// TIA Portal project "杨村程序" (V15.1)

(* hardware
DEVICE "S71500/ET200MP station_1"  S7-1500 station
   slot 0: "导轨_0"  Rack  6ES7 590-1***0-0AA0
   slot 1: "PLC_1"  CPU 1511-1 PN  6ES7 511-1AK02-0AB0  V2.6
      slot 3: "CPU 显示_1"  6ES7591-1AA00-0AA0
DEVICE "ET 200SP station_1"  ET 200SP-Station
   slot 0: "机架_0"  Rack  6ES5 710-8MAx1
   slot 0: "IO device_1"  IM 155-6 PN ST  6ES7 155-6AU01-0BN0  V4.1
   slot 1: "DI 16x24VDC ST_1"  DI 16x24VDC ST  6ES7 131-6BH01-0BA0  V0.0
      slot 1: "DI 16x24VDC ST_1"  DI 16x24VDC ST
   slot 2: "DI 16x24VDC ST_2"  DI 16x24VDC ST  6ES7 131-6BH01-0BA0  V0.0
      slot 1: "DI 16x24VDC ST_2"  DI 16x24VDC ST
   slot 3: "DI 16x24VDC ST_3"  DI 16x24VDC ST  6ES7 131-6BH01-0BA0  V0.0
      slot 1: "DI 16x24VDC ST_3"  DI 16x24VDC ST
   slot 4: "DI 16x24VDC ST_4"  DI 16x24VDC ST  6ES7 131-6BH01-0BA0  V0.0
      slot 1: "DI 16x24VDC ST_4"  DI 16x24VDC ST
   slot 5: "DQ 16x24VDC/0.5A ST_1"  DQ 16x24VDC/0.5A ST  6ES7 132-6BH01-0BA0  V0.0
      slot 1: "DQ 16x24VDC/0.5A ST_1"  DQ 16x24VDC/0.5A ST
   slot 6: "DQ 16x24VDC/0.5A ST_2"  DQ 16x24VDC/0.5A ST  6ES7 132-6BH01-0BA0  V0.0
      slot 1: "DQ 16x24VDC/0.5A ST_2"  DQ 16x24VDC/0.5A ST
   slot 7: "AI 8xI 2-,4-wire BA_1"  AI 8xI 2-,4-wire BA  6ES7 134-6GF00-0AA1  V1.0
      slot 1: "AI 8xI 2-,4-wire BA_1"  AI 8xI 2-,4-wire BA
   slot 8: "AI 8xI 2-,4-wire BA_2"  AI 8xI 2-,4-wire BA  6ES7 134-6GF00-0AA1  V1.0
      slot 1: "AI 8xI 2-,4-wire BA_2"  AI 8xI 2-,4-wire BA
   slot 9: "AI 8xI 2-,4-wire BA_3"  AI 8xI 2-,4-wire BA  6ES7 134-6GF00-0AA1  V1.0
      slot 1: "AI 8xI 2-,4-wire BA_3"  AI 8xI 2-,4-wire BA
   slot 10: "AI 8xI 2-,4-wire BA_4"  AI 8xI 2-,4-wire BA  6ES7 134-6GF00-0AA1  V1.0
      slot 1: "AI 8xI 2-,4-wire BA_4"  AI 8xI 2-,4-wire BA
   slot 11: "AQ 4xU/I ST_1"  AQ 4xU/I ST  6ES7 135-6HD00-0BA1  V1.1
      slot 1: "AQ 4xU/I ST_1"  AQ 4xU/I ST
   slot 12: "CM PtP_1"  CM PtP  6ES7 137-6AA00-0BA0  V1.0
      slot 1: "CM PtP_1"  CM PtP Sub
   slot 13: "服务器模块_1"  Server module  6ES7 193-6PA00-0AA0  V1.1
      slot 1: "服务器模块_1"  Server module
   slot 127: "BA 2xRJ45"  BA 2xRJ45  6ES7 193-6AR00-0AA0  V0.0
      slot 1: "Port_1"  X1 P1 R  6ES7 193-6AR00-0AA0  V0.0
      slot 2: "Port_2"  X1 P2 R  6ES7 193-6AR00-0AA0  V0.0
*)

// ===== PLC "PLC_1"  CPU 1511-1 PN =====

VAR_GLOBAL   // PLC tag table "默认变量表"
   "P1_HS" AT %IW8 : Int;
   "P2_HS" AT %IW10 : Int;
   "P3_GS" AT %IW12 : Int;
   "P4_GSFJK" AT %IW14 : Int;
   "P5_HSFJK" AT %IW16 : Int;
   "P6_GSCN" AT %IW18 : Int;
   "P7_HSCN" AT %IW20 : Int;
   "P1_能源站进站泵前压力" AT %MD100 : Real;
   "P2_能源站进站泵后压力" AT %MD104 : Real;
   "P3_能源站出站压力" AT %MD108 : Real;
   "P4_副井口供水压力" AT %MD112 : Real;
   "P5_副井口回水压力" AT %MD116 : Real;
   "P6_采暖供水压力" AT %MD120 : Real;
   "P7_采暖回水压力" AT %MD124 : Real;
   "T1_HS" AT %IW24 : Int;
   "T2_GS" AT %IW26 : Int;
   "T3_HSFJK1" AT %IW28 : Int;
   "T4_GSFJK1" AT %IW30 : Int;
   "T5_HSFJK2" AT %IW32 : Int;
   "T6_GSFJK2" AT %IW34 : Int;
   "T7_GSFJK" AT %IW36 : Int;
   "T8_HSFJK" AT %IW38 : Int;
   "T9_GSCN" AT %IW40 : Int;
   "T10_HSCN" AT %IW42 : Int;
   "T11_FJK_HJ" AT %IW44 : Int;
   "T12_SW_HJ" AT %IW46 : Int;
   "T1_能源站进站温度" AT %MD128 : Real;
   "T2_能源站出站温度" AT %MD132 : Real;
   "T3_副井口换热器一次进水" AT %MD136 : Real;
   "T4_副井口换热器一次出水" AT %MD140 : Real;
   "T5_副井口换热器二次进水" AT %MD144 : Real;
   "T6_副井口换热器二次出水" AT %MD148 : Real;
   "T7_副井口供水" AT %MD152 : Real;
   "T8_副井口回水" AT %MD156 : Real;
   "T9_采暖供水" AT %MD160 : Real;
   "T10_采暖回水" AT %MD164 : Real;
   "T11_副井口环境温度" AT %MD168 : Real;
   "T12_环境温度" AT %MD172 : Real;
   "隔离水泵运行频率" AT %MD176 : Real;
   "隔离水泵设定频率" AT %MD180 : Real;
   "MF1_ReadValue" AT %IW70 : Int;
   "System_Byte" AT %MB1 : Byte;
   "FirstScan" AT %M1.0 : Bool;
   "DiagStatusUpdate" AT %M1.1 : Bool;
   "AlwaysTRUE" AT %M1.2 : Bool;
   "AlwaysFALSE" AT %M1.3 : Bool;
   "Clock_Byte" AT %MB0 : Byte;
   "Clock_10Hz" AT %M0.0 : Bool;
   "Clock_5Hz" AT %M0.1 : Bool;
   "Clock_2.5Hz" AT %M0.2 : Bool;
   "Clock_2Hz" AT %M0.3 : Bool;
   "Clock_1.25Hz" AT %M0.4 : Bool;
   "Clock_1Hz" AT %M0.5 : Bool;
   "Clock_0.625Hz" AT %M0.6 : Bool;
   "Clock_0.5Hz" AT %M0.7 : Bool;
   "RM1_瞬时流量" AT %MD200 : Real;
   "RM1_瞬时热流量" AT %MD204 : Real;
   "RM1_累计热量" AT %MD208 : Real;
   "RM1_入口温度" AT %MD212 : Real;
   "RM1_出口温度" AT %MD216 : Real;
   "RM2_瞬时流量" AT %MD220 : Real;
   "RM2_瞬时热流量" AT %MD224 : Real;
   "RM2_累计热量" AT %MD228 : Real;
   "RM2_入口温度" AT %MD232 : Real;
   "RM2_出口温度" AT %MD236 : Real;
   "RM3_瞬时流量" AT %MD240 : Real;
   "RM3_瞬时热流量" AT %MD244 : Real;
   "RM3_累计热量" AT %MD248 : Real;
   "RM3_入口温度" AT %MD252 : Real;
   "RM3_出口温度" AT %MD256 : Real;
   "RM4_瞬时流量" AT %MD260 : Real;
   "RM4_瞬时热流量" AT %MD264 : Real;
   "RM4_累计热量" AT %MD268 : Real;
   "RM4_入口温度" AT %MD272 : Real;
   "RM4_出口温度" AT %MD276 : Real;
   "RM5_瞬时流量" AT %MD280 : Real;
   "RM5_瞬时热流量" AT %MD284 : Real;
   "RM5_累计热量" AT %MD288 : Real;
   "RM5_入口温度" AT %MD292 : Real;
   "RM5_出口温度" AT %MD296 : Real;
   "#1隔离泵手自状态反馈" AT %I0.0 : Bool;
   "#1隔离泵变频运行反馈" AT %I0.1 : Bool;
   "#1隔离泵变频故障反馈" AT %I0.2 : Bool;
   "#2隔离泵手自状态反馈" AT %I0.4 : Bool;
   "#2隔离泵软起运行反馈" AT %I0.5 : Bool;
   "#2隔离泵软起故障反馈" AT %I0.6 : Bool;
   "旁通电动阀手自状态反馈" AT %I1.0 : Bool;
   "#1电动阀全开反馈" AT %I1.1 : Bool;
   "#1电动阀全关反馈" AT %I1.2 : Bool;
   "#2电动阀全开反馈" AT %I1.3 : Bool;
   "#2电动阀全关反馈" AT %I1.4 : Bool;
   "#1进站水流开关状态" AT %I1.5 : Bool;
   "#2副井口水流开关状态" AT %I1.6 : Bool;
   "#3采暖水流开关状态" AT %I1.7 : Bool;
   "采暖循环泵手自状态反馈" AT %I2.0 : Bool;
   "#1采暖循环泵运行反馈" AT %I2.1 : Bool;
   "#2采暖循环泵运行反馈" AT %I2.2 : Bool;
   "#1采暖循环泵故障反馈" AT %I2.3 : Bool;
   "#2采暖循环泵故障反馈" AT %I2.4 : Bool;
   "副井口循环泵手自状态反馈" AT %I3.0 : Bool;
   "#1副井口循环泵运行反馈" AT %I3.1 : Bool;
   "#2副井口循环泵运行反馈" AT %I3.2 : Bool;
   "#3副井口循环泵运行反馈" AT %I3.3 : Bool;
   "供热补水泵手自状态反馈" AT %I4.0 : Bool;
   "#1供热补水泵运行反馈" AT %I4.1 : Bool;
   "#2供热补水泵运行反馈" AT %I4.2 : Bool;
   "矿区补水泵手自状态反馈" AT %I4.3 : Bool;
   "#1矿区补水泵运行反馈" AT %I4.4 : Bool;
   "#2矿区补水泵运行反馈" AT %I4.5 : Bool;
   "增压泵手自状态反馈" AT %I2.5 : Bool;
   "增加泵软起运行反馈" AT %I2.6 : Bool;
   "增压泵软起故障反馈" AT %I2.7 : Bool;
   "#1隔离水泵启停控制" AT %Q0.0 : Bool;
   "#2隔离水泵启停控制" AT %Q0.1 : Bool;
   "#1热泵机组旁通阀开控制" AT %Q0.2 : Bool;
   "#1热泵机组旁通阀关控制" AT %Q0.3 : Bool;
   "#2热泵机组旁通阀开控制" AT %Q0.4 : Bool;
   "#2热泵机组旁通阀关控制" AT %Q0.5 : Bool;
   "#1采暖泵启停控制" AT %Q0.6 : Bool;
   "#2采暖泵启停控制" AT %Q0.7 : Bool;
   "副井口#1采暖循环泵控制" AT %Q1.0 : Bool;
   "副井口#2采暖循环泵控制" AT %Q1.1 : Bool;
   "副井口#3采暖循环泵控制" AT %Q1.2 : Bool;
   "供热#1补水泵控制" AT %Q1.3 : Bool;
   "供热#2补水泵控制" AT %Q1.4 : Bool;
   "矿区#1补水泵控制" AT %Q1.5 : Bool;
   "矿区#2补水泵控制" AT %Q1.6 : Bool;
   "蜂鸣报警输出" AT %Q1.7 : Bool;
   "增压泵启停控制" AT %Q2.4 : Bool;
   "M_采暖#1泵手动启停" AT %M10.0 : Bool;
   "M_采暖#2泵手动启停" AT %M10.1 : Bool;
   "M_增压泵手动启停" AT %M10.2 : Bool;
   "M_副井口#1泵手动启停" AT %M10.3 : Bool;
   "M_副井口#2泵手动启停" AT %M10.4 : Bool;
   "M_副井口#3泵手动启停" AT %M10.5 : Bool;
   "M_隔离#1泵手动启停" AT %M10.6 : Bool;
   "M_隔离#2泵手动启停" AT %M10.7 : Bool;
   "M_供热补水#1泵手动启停" AT %M11.0 : Bool;
   "M_供热补水#2泵手动启停" AT %M11.1 : Bool;
   "M_矿区补水#1泵手动启停" AT %M11.2 : Bool;
   "M_矿区补水#2泵手动启停" AT %M11.3 : Bool;
   "M_旁通#1阀手动开关" AT %M11.4 : Bool;
   "M_旁通#2阀手动开关" AT %M11.5 : Bool;
   "M_电磁阀#1手动开关" AT %M11.6 : Bool;
   "S_循环水泵投入退出" AT %M2.0 : Bool;
   "水箱电磁阀启停控制" AT %Q3.4 : Bool;
   "Tag_2" AT %M20.1 : Bool;
   "Tag_3" AT %M20.0 : Bool;
   "Tag_4" AT %M20.2 : Bool;
   "Tag_5" AT %M20.3 : Bool;
   "Tag_6" AT %M20.4 : Bool;
   "Tag_7" AT %M20.5 : Bool;
   "Tag_8" AT %M20.6 : Bool;
   "Tag_9" AT %M20.7 : Bool;
   "Tag_10" AT %M21.0 : Bool;
   "Tag_11" AT %M21.1 : Bool;
   "Tag_12" AT %M21.2 : Bool;
   "Tag_13" AT %M21.3 : Bool;
   "Tag_14" AT %M21.4 : Bool;
   "Tag_15" AT %M21.5 : Bool;
   "Tag_16" AT %M21.6 : Bool;
   "Tag_17" AT %M21.7 : Bool;
   "Tag_18" AT %M22.0 : Bool;
   "Tag_19" AT %M22.1 : Bool;
   "Tag_20" AT %M22.2 : Bool;
   "Tag_21" AT %M22.3 : Bool;
   "Tag_22" AT %M22.4 : Bool;
   "Tag_23" AT %M22.5 : Bool;
   "Tag_24" AT %M22.6 : Bool;
   "Tag_25" AT %M22.7 : Bool;
   "Tag_26" AT %M23.0 : Bool;
   "Tag_27" AT %M23.1 : Bool;
   "Tag_28" AT %M23.2 : Bool;
   "Tag_29" AT %M23.3 : Bool;
   "Tag_30" AT %M23.4 : Bool;
   "Tag_31" AT %M23.5 : Bool;
   "系统运行天数" AT %MW90 : UInt;
   "系统运行小时" AT %MW92 : UInt;
   "系统运行分钟" AT %MW94 : UInt;
   "M_副井口排污阀手动开关" AT %M11.7 : Bool;
   "Tag_33" AT %M23.6 : Bool;
   "Tag_34" AT %M23.7 : Bool;
   "温度传感器上限" AT %MD310 : Real;
   "温度传感器下限" AT %MD314 : Real;
   "压力传感器上限" AT %MD318 : Real;
   "压力传感器下限" AT %MD322 : Real;
   "#1吸收式热泵启停指令" AT %MW326 : UInt;
   "#2吸收式热泵启停指令" AT %MW328 : UInt;
   "M_热泵 #1手动开关" AT %M12.0 : Bool;
   "M_热泵 #2手动开关" AT %M12.1 : Bool;
   "Tag_1" AT %M24.0 : Bool;
   "Tag_35" AT %M24.1 : Bool;
   "Tag_36" AT %M24.2 : Bool;
   "Tag_37" AT %M24.3 : Bool;
   "变频器频率上限" AT %MD330 : Real;
   "变频器频率下限" AT %MD334 : Real;
   "MF1_WriteFValue" AT %QW4 : Int;
   "#1热泵热网水进口温度" AT %MD340 : Real;
   "#1热泵热网水出口温度" AT %MD344 : Real;
   "#1热泵热源水进口温度" AT %MD348 : Real;
   "#1热泵热源水出口温度" AT %MD352 : Real;
   "#1热泵驱动热水进口温度" AT %MD356 : Real;
   "#1热泵驱动热水出口温度" AT %MD360 : Real;
   "#2热泵热网水进口温度" AT %MD364 : Real;
   "#2热泵热网水出口温度" AT %MD368 : Real;
   "#2热泵热源水进口温度" AT %MD372 : Real;
   "#2热泵热源水出口温度" AT %MD376 : Real;
   "#2热泵驱动热水进口温度" AT %MD380 : Real;
   "#2热泵驱动热水出口温度" AT %MD384 : Real;
   "国焦侧供水温度" AT %MD388 : Real;
   "国焦侧回水温度" AT %MD392 : Real;
   "国焦侧氨水进水温度" AT %MD396 : Real;
   "国焦侧氨水回水温度" AT %MD400 : Real;
   "国焦侧蒸汽瞬时流量" AT %MD404 : Real;
   "供热补水压力上限" AT %MD408 : Real;
   "供热补水压力下限" AT %MD412 : Real;
   "矿区补水压力上限" AT %MD416 : Real;
   "矿区补水压力下限" AT %MD420 : Real;
   "M_补水泵手自投入退出" AT %M2.1 : Bool;
   "Tag_38" AT %M24.5 : Bool;
   "Tag_39" AT %M24.6 : Bool;
   "Tag_40" AT %M24.7 : Bool;
   "Tag_41" AT %M25.0 : Bool;
   "Tag_42" AT %M25.1 : Bool;
   "Tag_43" AT %M25.2 : Bool;
   "Tag_44" AT %M25.3 : Bool;
   "Tag_45" AT %M25.4 : Bool;
   "补水参数设置错误" AT %M50.6 : Bool;
   "水箱液位" AT %MD424 : Real;
   "H_Yewei" AT %IW56 : Int;
   "电加热管道AP7电源合闸反馈" AT %I3.4 : Bool;
   "电加热管道AP7电源分闸反馈" AT %I3.5 : Bool;
   "电加热管道AP7电源故障反馈" AT %I3.6 : Bool;
   "电加热管道AP8电源合闸反馈" AT %I5.4 : Bool;
   "电加热管道AP8电源分闸反馈" AT %I5.5 : Bool;
   "电加热管道AP8电源故障反馈" AT %I5.6 : Bool;
   "#2采暖排污阀关控制" AT %Q3.3 : Bool;
   "#2采暖排污阀开控制" AT %Q3.2 : Bool;
   "#1副井口排污阀关控制" AT %Q3.1 : Bool;
   "#1副井口排污阀开控制" AT %Q3.0 : Bool;
   "#1副井口排污阀开反馈" AT %I5.0 : Bool;
   "M_采暖排污阀手动开关" AT %M12.2 : Bool;
   "Tag_47" AT %M25.5 : Bool;
   "Tag_48" AT %M25.6 : Bool;
   "Tag_49" AT %M25.7 : Bool;
   "Tag_50" AT %M26.0 : Bool;
   "报警_水箱液位低" AT %M50.0 : Bool;
   "报警_水箱液位高" AT %M50.1 : Bool;
   "供热补水泵#1投入" AT %M3.1 : Bool;
   "modbus_Step" AT %MW56 : UInt;
   "供热补水泵#2投入" AT %M3.2 : Bool;
   "矿区补水泵#1投入" AT %M3.3 : Bool;
   "矿区补水泵#2投入" AT %M3.4 : Bool;
   "#1副井口排污阀关反馈" AT %I5.1 : Bool;
   "#2采暖排污阀开反馈" AT %I5.2 : Bool;
   "#2采暖排污阀关反馈" AT %I5.3 : Bool;
   "#1热泵启动控制" AT %Q2.0 : Bool;
   "#1热泵急停控制" AT %Q2.1 : Bool;
   "#2热泵启动控制" AT %Q2.2 : Bool;
   "#2热泵急停控制" AT %Q2.3 : Bool;
   "P1_能源站进站泵前压力_工程值" AT %MD428 : Real;
   "P2_能源站进站泵后压力_工程值" AT %MD432 : Real;
   "P3_能源站出站压力_工程值" AT %MD436 : Real;
   "P4_副井口供水压力_工程值" AT %MD440 : Real;
   "P5_副井口回水压力_工程值" AT %MD444 : Real;
   "P6_采暖供水压力_工程值" AT %MD448 : Real;
   "P7_采暖回水压力_工程值" AT %MD452 : Real;
   "T1_能源站进站温度_工程值" AT %MD456 : Real;
   "T2_能源站出站温度_工程值" AT %MD460 : Real;
   "T3_副井口换热器一次进水_工程值" AT %MD464 : Real;
   "T4_副井口换热器一次出水_工程值" AT %MD468 : Real;
   "T5_副井口换热器二次进水_工程值" AT %MD472 : Real;
   "T6_副井口换热器二次出水_工程值" AT %MD476 : Real;
   "T7_副井口供水_工程值" AT %MD480 : Real;
   "T8_副井口回水_工程值" AT %MD484 : Real;
   "T9_采暖供水_工程值" AT %MD488 : Real;
   "T10_采暖回水_工程值" AT %MD492 : Real;
   "T11_副井口环境温度_工程值" AT %MD496 : Real;
   "T12_环境温度_工程值" AT %MD500 : Real;
   "水箱液位_工程值" AT %MD504 : Real;
   "隔离水泵运行频率_工程值" AT %MD508 : Real;
   "M_电动阀手自投入退出" AT %M2.2 : Bool;   // 0-手动 1-自动
   "S_热泵投入退出" AT %M2.3 : Bool;
   "S_补水泵投入退出" AT %M2.4 : Bool;
   "S_电动阀投入退出" AT %M2.5 : Bool;
   "供热#1补水泵故障" AT %M50.2 : Bool;
   "供热#2补水泵故障" AT %M50.3 : Bool;
   "矿区#1补水泵故障" AT %M50.4 : Bool;
   "矿区#2补水泵故障" AT %M50.5 : Bool;
   "modbus_temp" AT %MW60 : Word;
   "Modbus_Tmp2" AT %MW62 : Word;
   "#1热泵热网水进口压力" AT %MD512 : Real;
   "#1热泵热网水出口压力" AT %MD516 : Real;
   "#1热泵热源水进口压力" AT %MD520 : Real;
   "#1热泵热源水出口压力" AT %MD524 : Real;
   "#1热泵驱动热水进口压力" AT %MD528 : Real;
   "#1热泵驱动热水出口压力" AT %MD532 : Real;
   "#2热泵热网水进口压力" AT %MD536 : Real;
   "#2热泵热网水出口压力" AT %MD540 : Real;
   "#2热泵热源水进口压力" AT %MD544 : Real;
   "#2热泵热源水出口压力" AT %MD548 : Real;
   "#2热泵驱动热水进口压力" AT %MD552 : Real;
   "#2热泵驱动热水出口压力" AT %MD556 : Real;
   "#1吸收式热泵故障值" AT %MW96 : UInt;
   "#2吸收式热泵故障值" AT %MW98 : Word;
   "#1吸收式热泵运作状态" AT %M12.3 : Bool;
   "#2吸收式热泵运作状态" AT %M12.4 : Bool;
   "Tag_46" AT %M26.1 : Bool;
   "Tag_51" AT %M26.2 : Bool;
   "Tag_52" AT %M26.3 : Bool;
   "Tag_53" AT %M26.4 : Bool;
   "Tag_54" AT %M26.5 : Bool;
   "Tag_55" AT %M26.7 : Bool;
   "RM1_瞬时流量_记录" AT %MD560 : Real;
   "RM2_瞬时流量_记录" AT %MD564 : Real;
   "RM3_瞬时流量_记录" AT %MD568 : Real;
   "RM4_瞬时流量_记录" AT %MD572 : Real;
   "RM5_瞬时流量_记录" AT %MD576 : Real;
   "系统故障" AT %M40.0 : Bool;
   "系统报警" AT %M40.1 : Bool;
   "故障手动复位" AT %M4.0 : Bool;
   "Tag_32" AT %M27.0 : Bool;
   "Tag_56" AT %M27.1 : Bool;
   "Tag_57" AT %M27.2 : Bool;
   "Tag_58" AT %T1 : Timer;
END_VAR

TYPE "RM_STRUCT"
   STRUCT
      热流量 : Real;
      累计热量整数 : UDInt;
      累计热量小数 : Real;
      入口温度 : UInt;
      出口温度 : UInt;
   END_STRUCT;
END_TYPE

TYPE "RMotor_STRUCT"
   STRUCT
      AI0 : Int;
      AI1 : Int;
      AI2 : Int;
      AI3 : Int;
      AI4 : Int;
      AI5 : Int;
      AI6 : Int;
      AI7 : Int;
      AI8 : Int;
      AI9 : Int;
   END_STRUCT;
END_TYPE

TYPE "RMotor_State"
   STRUCT
      State : Array[0..2] of Word;
   END_STRUCT;
END_TYPE

DATA_BLOCK "DB_MasterData"   // DB1
{ S7_Optimized_Access := 'FALSE' }
VERSION : 0.1
   VAR
      M1_Data1 : Array[0..1] of Word;
      M1_Data2 : "RM_STRUCT";
      Master_Done_Marks : Array[0..19] of Bool;
      Master_Error_Marks : Array[0..19] of Bool;
      Master_Busy_Marks : Array[0..19] of Bool;
      Master_Status : Array[0..19] of Word;
      Modbus_Step : USInt;
      CommLoad_Done : Bool;
      CommLoad_ERROR : Bool;
      CommLoad_STATUS : Word;
      M2_Data1 : Array[0..1] of Word;
      M2_Data2 : "RM_STRUCT";
      M3_Data1 : Array[0..1] of Word;
      M3_Data2 : "RM_STRUCT";
      M4_Data1 : Array[0..1] of Word;
      M4_Data2 : "RM_STRUCT";
      M5_Data1 : Array[0..1] of Word;
      M5_Data2 : "RM_STRUCT";
      RMoter1_AIData1 : Array[0..3] of Int;   // 温度
      RMoter2_AIData1 : Array[0..3] of Int;   // 温度
      RMoter1_AIData2 : Array[0..1] of Int;   // 温度
      RMoter2_AIData2 : Array[0..1] of Int;   // 温度
      RMoter1_AIData3 : Array[0..5] of Int;   // 压力
      RMoter2_AIData3 : Array[0..5] of Int;   // 压力
      RMoter1_AIData4 : Array[0..1] of Word;   // 状态
      RMoter2_AIData4 : Array[0..1] of Word;   // 状态
   END_VAR
BEGIN
END_DATA_BLOCK

DATA_BLOCK "中间变量值"   // DB2
{ S7_Optimized_Access := 'TRUE' }
VERSION : 0.1
   VAR
      P1_NORM_REAL : Real;
      P2_NORM_REAL : Real;
      P3_NORM_REAL : Real;
      P4_NORM_REAL : Real;
      P5_NORM_REAL : Real;
      P6_NORM_REAL : Real;
      P7_NORM_REAL : Real;
      T1_NORM_REAL : Real;
      T2_NORM_REAL : Real;
      T3_NORM_REAL : Real;
      T4_NORM_REAL : Real;
      T5_NORM_REAL : Real;
      T6_NORM_REAL : Real;
      T7_NORM_REAL : Real;
      T8_NORM_REAL : Real;
      T9_NORM_REAL : Real;
      T10_NORM_REAL : Real;
      T11_NORM_REAL : Real;
      T12_NORM_REAL : Real;
      MF1_NORM_REAL : Real;
      MF1_NORM1_REAL : Real;
      RM1_T1_入口 : Real;
      RM1_T2_出口 : Real;
      RM2_T1_入口 : Real;
      RM2_T2_出口 : Real;
      RM3_T1_入口 : Real;
      RM3_T2_出口 : Real;
      RM4_T1_入口 : Real;
      RM4_T2_出口 : Real;
      RM5_T1_入口 : Real;
      RM5_T2_出口 : Real;
      RM_TMP_REAL_1 : Real;
      RM_TMP_REAL_2 : Real;
      RM_TMP_REAL_3 : Real;
      RM_TMP_REAL_4 : Real;
      RM_TMP_REAL_5 : Real;
      H_TMP_REAL : Real;
      "V_M_Q0.0" : Bool;   // #1隔离泵控制输出中间变量
      "V_M_Q0.1" : Bool;   // #2隔离泵控制输出中间变量
      "V_M_Q0.2" : Bool;   // #1旁通阀开输出中间变量
      "V_M_Q0.3" : Bool;   // #1旁通阀关输出中间变量
      "V_M_Q0.4" : Bool;   // #2旁通阀开输出中间变量
      "V_M_Q0.5" : Bool;   // #2旁通阀关输出中间变量
      "V_M_Q0.6" : Bool;   // #1采暖泵控制输出中间变量
      "V_M_Q0.7" : Bool;   // #2采暖泵控制输出中间变量
      "V_M_Q1.0" : Bool;   // #1副井口泵控制输出中间变量
      "V_M_Q1.1" : Bool;   // #2副井口泵控制输出中间变量
      "V_M_Q1.2" : Bool;   // #3副井口泵控制输出中间变量
      "V_M_Q1.3" : Bool;   // #1供热补水泵控制输出中间变量
      "V_M_Q1.4" : Bool;   // #2供热补水泵控制输出中间变量
      "V_M_Q1.5" : Bool;   // #1矿区补水泵控制输出中间变量
      "V_M_Q1.6" : Bool;   // #2矿区补水泵控制输出中间变量
      "V_M_Q1.7" : Bool;   // 报警蜂鸣器控制输出中间变量
      "V_M_Q2.0" : Bool;   // #1吸收式热泵启动输出中间变量
      "V_M_Q2.1" : Bool;   // #1吸收式热泵停止输出中间变量
      "V_M_Q2.2" : Bool;   // #2吸收式热泵启动输出中间变量
      "V_M_Q2.3" : Bool;   // #2吸收式热泵停止输出中间变量
      "V_M_Q2.4" : Bool;   // 增压泵控制输出中间变量
      "V_M_Q3.0" : Bool;   // #1副井口排污阀开控制输出中间变量
      "V_M_Q3.1" : Bool;   // #1副井口排污阀关控制输出中间变量
      "V_M_Q3.2" : Bool;   // #2采暖排污阀开控制输出中间变量
      "V_M_Q3.3" : Bool;   // #2采暖排污阀关控制输出中间变量
      "V_M_Q3.4" : Bool;   // 电磁阀#1控制输出中间变量
      V_M_RM1 : Bool;   // 吸收式热泵#1控制输出中间变量
      V_M_RM2 : Bool;   // 吸收式热泵#2控制输出中间变量
      RMotor1_T1 : Real;   // #1热泵驱动热水进口温度读取值
      RMotor1_T2 : Real;   // #1热泵驱动热水出口温度读取值
      RMotor2_T1 : Real;   // #2热泵驱动热水进口温度读取值
      RMotor2_T2 : Real;   // #2热泵驱动热水出口温度读取值
      RMotor1_AI0 : Real;   // #1热泵热网水进口温度读取值
      RMotor1_AI1 : Real;   // #1热泵热网水出口温度读取值
      RMotor1_AI2 : Real;   // #1热泵热源水进口温度读取值
      RMotor1_AI3 : Real;   // #1热泵热源水出口温度读取值
      RMotor2_AI0 : Real;   // #2热泵热网水进口温度读取值
      RMotor2_AI1 : Real;   // #2热泵热网水出口温度读取值
      RMotor2_AI2 : Real;   // #2热泵热源水进口温度读取值
      RMotor2_AI3 : Real;   // #2热泵热源水出口温度读取值
      RMotor1_P1 : Real;
      RMotor1_P2 : Real;
      RMotor1_P3 : Real;
      RMotor1_P4 : Real;
      RMotor1_P5 : Real;
      RMotor1_P6 : Real;
      RMotor2_P1 : Real;
      RMotor2_P2 : Real;
      RMotor2_P3 : Real;
      RMotor2_P4 : Real;
      RMotor2_P5 : Real;
      RMotor2_P6 : Real;
      补水泵控制高限位延时换算s : DWord := 0;
      补水泵控制低限位延时换算s : DWord := 0;
      排污阀控制延时换算s : DWord := 0;
      系统故障数组计算值 : Bool;
      系统报警数组计算值 : Bool;
      压力异常报警延时换算s : DWord := 0;
      温度异常报警延时换算s : DWord := 0;
      采暖泵压差异常报警延时换算s : DWord := 0;
      系统报警数组中间值 : Array[0..31] of Bool;
      一网采暖泵压力差值 : Real;
   END_VAR
BEGIN
END_DATA_BLOCK

DATA_BLOCK "DB_参数设置"   // DB5
{ S7_Optimized_Access := 'FALSE' }
VERSION : 0.1
   VAR
      水箱液位低报警设值 : Real := 0.5;
      水箱液位高报警设值 : Real := 2.6;
      矿区补水压力下限 : Real := 0.3;
      矿区补水压力上限 : Real := 0.6;
      供热补水压力下限 : Real := 0.2;
      供热补水压力上限 : Real := 0.4;
      变频器频率下限 : Real;
      变频器频率上限 : Real := 50.0;
      隔离水泵设定频率 : Real := 50.0;
      能源站进站温度T1上限 : Real := 200.0;
      能源站进站温度T1下限 : Real := -50.0;
      能源站出站温度T2上限 : Real := 200.0;
      能源站出站温度T2下限 : Real := -50.0;
      副井口一次进水温度T3上限 : Real := 200.0;
      副井口一次进水温度T3下限 : Real := -50.0;
      副井口一次出水温度T4上限 : Real := 200.0;
      副井口一次出水温度T4下限 : Real := -50.0;
      副井口二次进水温度T5上限 : Real := 200.0;
      副井口二次进水温度T5下限 : Real := -50.0;
      副井口二次出水温度T6上限 : Real := 200.0;
      副井口二次出水温度T6下限 : Real := -50.0;
      副井口供水温度T7上限 : Real := 200.0;
      副井口供水温度T7下限 : Real := -50.0;
      副井口回水温度T8上限 : Real := 200.0;
      副井口回水温度T8下限 : Real := -50.0;
      采暖供水温度T9上限 : Real := 200.0;
      采暖供水温度T9下限 : Real := -50.0;
      采暖回水温度T10上限 : Real := 200.0;
      采暖回水温度T10下限 : Real := -50.0;
      副井口环境温度T11上限 : Real := 200.0;
      副井口环境温度T11下限 : Real := -50.0;
      环境温度T12上限 : Real := 200.0;
      环境温度T12下限 : Real := -50.0;
      能源站进站压力P1上限 : Real := 2.4;
      能源站进站压力P1下限 : Real := -0.1;
      能源站进站泵后压力P2上限 : Real := 2.4;
      能源站进站泵后压力P2下限 : Real := -0.1;
      能源站出站压力P3上限 : Real := 2.4;
      能源站出站压力P3下限 : Real := -0.1;
      副井口供水压力P4上限 : Real := 2.4;
      副井口供水压力P4下限 : Real := -0.1;
      副井口回水压力P5上限 : Real := 2.4;
      副井口回水压力P5下限 : Real := -0.1;
      采暖供水压力P6上限 : Real := 2.4;
      采暖供水压力P6下限 : Real := -0.1;
      采暖回水压力P7上限 : Real := 2.4;
      采暖回水压力P7下限 : Real := -0.1;
      补水箱液位上限 : Real := 2.8;
      补水箱液位下限 : Real;
      T1修正值 : Real;
      T2修正值 : Real;
      T3修正值 : Real;
      T4修正值 : Real;
      T5修正值 : Real;
      T6修正值 : Real;
      T7修正值 : Real;
      T8修正值 : Real;
      T9修正值 : Real;
      T10修正值 : Real;
      T11修正值 : Real;
      T12修正值 : Real;
      P1修正值 : Real;
      P2修正值 : Real;
      P3修正值 : Real;
      P4修正值 : Real;
      P5修正值 : Real;
      P6修正值 : Real;
      P7修正值 : Real;
      液位修正值 : Real := 1.06;
      频率修正值 : Real;
      补水泵高位延时 : DWord := 3;
      补水泵低位延时 : DWord := 3;
      "副井口#1排污阀开压力值" : Real := 0.4;
      "副井口#1排污阀关压力值" : Real := 0.3;
      "采暖#2排污阀开压力值" : Real := 0.78;
      "采暖#2排污阀关压力值" : Real := 0.56;
      排污阀控制延时 : DWord := 3;
      补水箱电磁阀开液位 : Real := 2.0;
      补水箱电磁阀关液位 : Real := 2.65;
      系统报警列表 : Array[0..32] of Bool;
      系统故障列表 : Array[0..32] of Bool;
      P1异常报警上下限值 : Array[0..1] of Real;
      P2异常报警上下限值 : Array[0..1] of Real;
      P3异常报警上下限值 : Array[0..1] of Real;
      P4异常报警上下限值 : Array[0..1] of Real;
      P5异常报警上下限值 : Array[0..1] of Real;
      P6异常报警上下限值 : Array[0..1] of Real;
      P7异常报警上下限值 : Array[0..1] of Real;
      副井口温度异常报警设置 : Array[0..1] of Real;
      采暖回水温度异常报警设置 : Array[0..1] of Real;
      一网进站温度异常报警设值 : Array[0..1] of Real;
      采暖泵压差上限设值 : Real := 1.0;
      压力异常报警延时 : UInt := 3;
      温度异常报警延时 : UInt := 3;
      采暖泵压差异常报警延时 : UInt := 3;
   END_VAR
BEGIN
   P1异常报警上下限值[1] := -0.1;   // 下限
   P2异常报警上下限值[1] := -0.1;   // 下限
   P3异常报警上下限值[1] := -0.1;   // 下限
   P4异常报警上下限值[1] := -0.1;   // 下限
   P1异常报警上下限值[0] := 1.0;   // 上限
   P2异常报警上下限值[0] := 1.0;   // 上限
   P3异常报警上下限值[0] := 1.0;   // 上限
   P4异常报警上下限值[0] := 1.0;   // 上限
   P5异常报警上下限值[0] := 1.0;   // 上限
   P5异常报警上下限值[1] := -0.1;   // 下限
   P6异常报警上下限值[0] := 1.0;   // 上限
   P6异常报警上下限值[1] := -0.1;   // 下限
   P7异常报警上下限值[0] := 1.0;   // 上限
   P7异常报警上下限值[1] := -0.1;   // 下限
   副井口温度异常报警设置[0] := 60.0;   // 上限
   采暖回水温度异常报警设置[0] := 90.0;   // 上限
   一网进站温度异常报警设值[0] := 110.0;   // 上限
   // 系统报警列表[0] : 水箱液位高报警
   // 系统报警列表[1] : 水箱液位低报警
   // 系统报警列表[2] : 补水压力参数设置错误报警
   // 系统故障列表[0] : 矿区补水泵#1故障
   // 系统故障列表[1] : 矿区补水泵#2故障
   // 系统故障列表[2] : 供热补水泵#1故障
   // 系统故障列表[3] : 供热补水泵#2故障
   // 副井口温度异常报警设置[1] : 下限
   // 采暖回水温度异常报警设置[1] : 下限
   // 一网进站温度异常报警设值[1] : 下限
   // 系统报警列表[3] : 进站泵前压力P1异常报警
   // 系统报警列表[4] : 进站泵后压力P2异常报警
   // 系统报警列表[5] : 出站压力P3异常报警
   // 系统报警列表[6] : 副井口供水压力P4异常报警
   // 系统报警列表[7] : 副井口回水压力P5异常报警
   // 系统报警列表[8] : 采暖供水压力P6异常报警
   // 系统报警列表[9] : 采暖回水压力P7异常报警
   // 系统报警列表[10] : 副井口回水温度T8异常报警
   // 系统报警列表[11] : 采暖回水温度T10异常报警
   // 系统报警列表[12] : 一网进站温度T1异常报警
   // 系统报警列表[13] : 一网采暖泵压差异常报警
   // 系统故障列表[4] : 吸收式热泵#1故障
   // 系统故障列表[5] : 吸收式热泵#2故障
   // 系统故障列表[6] : 副井口循环泵#1故障
   // 系统故障列表[7] : 副井口循环泵#2故障
   // 系统故障列表[8] : 副井口循环泵#3故障
   // 系统故障列表[9] : 国焦焦化侧故障
END_DATA_BLOCK

DATA_BLOCK "fb_modbus通讯_DB"   // DB8
{ S7_Optimized_Access := 'TRUE' }
VERSION : 0.1
// stored: InstanceOfName fb_modbus通讯
"fb_modbus通讯"
BEGIN
END_DATA_BLOCK

DATA_BLOCK "test_DB"   // DB19
{ S7_Optimized_Access := 'FALSE' }
VERSION : 0.1
   VAR
      MData : Array[0..20] of Word;
      MData_1 : Array[0..20] of Int;
   END_VAR
BEGIN
END_DATA_BLOCK

// folder: System blocks/Program resources

DATA_BLOCK "IEC_Timer_0_DB"   // DB3
{ S7_Optimized_Access := 'TRUE' }
AUTHOR : Simatic
FAMILY : IEC
NAME : IEC_TMR
VERSION : 1.0
// stored: InstanceOfName IEC_TIMER
"IEC_TIMER"
BEGIN
END_DATA_BLOCK

DATA_BLOCK "IEC_Timer_1_DB"   // DB4
{ S7_Optimized_Access := 'TRUE' }
AUTHOR : Simatic
FAMILY : IEC
NAME : IEC_TMR
VERSION : 1.0
// stored: InstanceOfName IEC_TIMER
"IEC_TIMER"
BEGIN
END_DATA_BLOCK

DATA_BLOCK "IEC_Timer_2_DB_1"   // DB6
{ S7_Optimized_Access := 'TRUE' }
AUTHOR : Simatic
FAMILY : IEC
NAME : IEC_TMR
VERSION : 1.0
// stored: InstanceOfName IEC_TIMER
"IEC_TIMER"
BEGIN
END_DATA_BLOCK

DATA_BLOCK "IEC_Timer_2_DB"   // DB7
{ S7_Optimized_Access := 'TRUE' }
AUTHOR : Simatic
FAMILY : IEC
NAME : IEC_TMR
VERSION : 1.0
// stored: InstanceOfName IEC_TIMER
"IEC_TIMER"
BEGIN
END_DATA_BLOCK

DATA_BLOCK "IEC_Timer_3_DB"   // DB9
{ S7_Optimized_Access := 'TRUE' }
AUTHOR : Simatic
FAMILY : IEC
NAME : IEC_TMR
VERSION : 1.0
// stored: InstanceOfName IEC_TIMER
"IEC_TIMER"
BEGIN
END_DATA_BLOCK

DATA_BLOCK "IEC_Timer_0_DB_2"   // DB10
{ S7_Optimized_Access := 'TRUE' }
AUTHOR : Simatic
FAMILY : IEC
NAME : IEC_TMR
VERSION : 1.0
// stored: InstanceOfName IEC_TIMER
"IEC_TIMER"
BEGIN
END_DATA_BLOCK

DATA_BLOCK "IEC_Timer_0_DB_3"   // DB11
{ S7_Optimized_Access := 'TRUE' }
AUTHOR : Simatic
FAMILY : IEC
NAME : IEC_TMR
VERSION : 1.0
// stored: InstanceOfName IEC_TIMER
"IEC_TIMER"
BEGIN
END_DATA_BLOCK

DATA_BLOCK "IEC_Timer_2_DB_2"   // DB12
{ S7_Optimized_Access := 'TRUE' }
AUTHOR : Simatic
FAMILY : IEC
NAME : IEC_TMR
VERSION : 1.0
// stored: InstanceOfName IEC_TIMER
"IEC_TIMER"
BEGIN
END_DATA_BLOCK

DATA_BLOCK "IEC_Timer_2_DB_3"   // DB13
{ S7_Optimized_Access := 'TRUE' }
AUTHOR : Simatic
FAMILY : IEC
NAME : IEC_TMR
VERSION : 1.0
// stored: InstanceOfName IEC_TIMER
"IEC_TIMER"
BEGIN
END_DATA_BLOCK

DATA_BLOCK "IEC_Timer_2_DB_4"   // DB14
{ S7_Optimized_Access := 'TRUE' }
AUTHOR : Simatic
FAMILY : IEC
NAME : IEC_TMR
VERSION : 1.0
// stored: InstanceOfName IEC_TIMER
"IEC_TIMER"
BEGIN
END_DATA_BLOCK

DATA_BLOCK "IEC_Timer_1_DB_1"   // DB15
{ S7_Optimized_Access := 'TRUE' }
AUTHOR : Simatic
FAMILY : IEC
NAME : IEC_TMR
VERSION : 1.0
// stored: InstanceOfName IEC_TIMER
"IEC_TIMER"
BEGIN
END_DATA_BLOCK

DATA_BLOCK "IEC_Timer_1_DB_2"   // DB18
{ S7_Optimized_Access := 'TRUE' }
AUTHOR : Simatic
FAMILY : IEC
NAME : IEC_TMR
VERSION : 1.0
// stored: InstanceOfName IEC_TIMER
"IEC_TIMER"
BEGIN
END_DATA_BLOCK

DATA_BLOCK "IEC_Timer_1_DB_3"   // DB20
{ S7_Optimized_Access := 'TRUE' }
AUTHOR : Simatic
FAMILY : IEC
NAME : IEC_TMR
VERSION : 1.0
// stored: InstanceOfName IEC_TIMER
"IEC_TIMER"
BEGIN
END_DATA_BLOCK

DATA_BLOCK "IEC_Timer_1_DB_4"   // DB21
{ S7_Optimized_Access := 'TRUE' }
AUTHOR : Simatic
FAMILY : IEC
NAME : IEC_TMR
VERSION : 1.0
// stored: InstanceOfName IEC_TIMER
"IEC_TIMER"
BEGIN
END_DATA_BLOCK

DATA_BLOCK "IEC_Timer_4DB1"   // DB22
{ S7_Optimized_Access := 'TRUE' }
AUTHOR : Simatic
FAMILY : IEC
NAME : IEC_TMR
VERSION : 1.0
// stored: InstanceOfName IEC_TIMER
"IEC_TIMER"
BEGIN
END_DATA_BLOCK

DATA_BLOCK "IEC_Timer_4_DB_1"   // DB23
{ S7_Optimized_Access := 'TRUE' }
AUTHOR : Simatic
FAMILY : IEC
NAME : IEC_TMR
VERSION : 1.0
// stored: InstanceOfName IEC_TIMER
"IEC_TIMER"
BEGIN
END_DATA_BLOCK

DATA_BLOCK "IEC_Timer_4DB2"   // DB24
{ S7_Optimized_Access := 'TRUE' }
AUTHOR : Simatic
FAMILY : IEC
NAME : IEC_TMR
VERSION : 1.0
// stored: InstanceOfName IEC_TIMER
"IEC_TIMER"
BEGIN
END_DATA_BLOCK

DATA_BLOCK "IEC_Timer_4DB3"   // DB25
{ S7_Optimized_Access := 'TRUE' }
AUTHOR : Simatic
FAMILY : IEC
NAME : IEC_TMR
VERSION : 1.0
// stored: InstanceOfName IEC_TIMER
"IEC_TIMER"
BEGIN
END_DATA_BLOCK

DATA_BLOCK "IEC_Timer_4DB4"   // DB26
{ S7_Optimized_Access := 'TRUE' }
AUTHOR : Simatic
FAMILY : IEC
NAME : IEC_TMR
VERSION : 1.0
// stored: InstanceOfName IEC_TIMER
"IEC_TIMER"
BEGIN
END_DATA_BLOCK

DATA_BLOCK "IEC_Timer_4DB5"   // DB27
{ S7_Optimized_Access := 'TRUE' }
AUTHOR : Simatic
FAMILY : IEC
NAME : IEC_TMR
VERSION : 1.0
// stored: InstanceOfName IEC_TIMER
"IEC_TIMER"
BEGIN
END_DATA_BLOCK

DATA_BLOCK "IEC_Timer_4DB6"   // DB28
{ S7_Optimized_Access := 'TRUE' }
AUTHOR : Simatic
FAMILY : IEC
NAME : IEC_TMR
VERSION : 1.0
// stored: InstanceOfName IEC_TIMER
"IEC_TIMER"
BEGIN
END_DATA_BLOCK

DATA_BLOCK "IEC_Timer_4DB7"   // DB29
{ S7_Optimized_Access := 'TRUE' }
AUTHOR : Simatic
FAMILY : IEC
NAME : IEC_TMR
VERSION : 1.0
// stored: InstanceOfName IEC_TIMER
"IEC_TIMER"
BEGIN
END_DATA_BLOCK

DATA_BLOCK "IEC_Timer_5DB1"   // DB30
{ S7_Optimized_Access := 'TRUE' }
AUTHOR : Simatic
FAMILY : IEC
NAME : IEC_TMR
VERSION : 1.0
// stored: InstanceOfName IEC_TIMER
"IEC_TIMER"
BEGIN
END_DATA_BLOCK

DATA_BLOCK "IEC_Timer_5DB2"   // DB31
{ S7_Optimized_Access := 'TRUE' }
AUTHOR : Simatic
FAMILY : IEC
NAME : IEC_TMR
VERSION : 1.0
// stored: InstanceOfName IEC_TIMER
"IEC_TIMER"
BEGIN
END_DATA_BLOCK

DATA_BLOCK "IEC_Timer_5DB3"   // DB32
{ S7_Optimized_Access := 'TRUE' }
AUTHOR : Simatic
FAMILY : IEC
NAME : IEC_TMR
VERSION : 1.0
// stored: InstanceOfName IEC_TIMER
"IEC_TIMER"
BEGIN
END_DATA_BLOCK

DATA_BLOCK "IEC_Timer_4DB8"   // DB33
{ S7_Optimized_Access := 'TRUE' }
AUTHOR : Simatic
FAMILY : IEC
NAME : IEC_TMR
VERSION : 1.0
// stored: InstanceOfName IEC_TIMER
"IEC_TIMER"
BEGIN
END_DATA_BLOCK

DATA_BLOCK "IEC_Timer_4DB9"   // DB34
{ S7_Optimized_Access := 'TRUE' }
AUTHOR : Simatic
FAMILY : IEC
NAME : IEC_TMR
VERSION : 1.0
// stored: InstanceOfName IEC_TIMER
"IEC_TIMER"
BEGIN
END_DATA_BLOCK

DATA_BLOCK "IEC_Timer_4DB10"   // DB35
{ S7_Optimized_Access := 'TRUE' }
AUTHOR : Simatic
FAMILY : IEC
NAME : IEC_TMR
VERSION : 1.0
// stored: InstanceOfName IEC_TIMER
"IEC_TIMER"
BEGIN
END_DATA_BLOCK

DATA_BLOCK "IEC_Timer_4DB11"   // DB36
{ S7_Optimized_Access := 'TRUE' }
AUTHOR : Simatic
FAMILY : IEC
NAME : IEC_TMR
VERSION : 1.0
// stored: InstanceOfName IEC_TIMER
"IEC_TIMER"
BEGIN
END_DATA_BLOCK

DATA_BLOCK "IEC_Timer_6DB_11"   // DB37
{ S7_Optimized_Access := 'TRUE' }
AUTHOR : Simatic
FAMILY : IEC
NAME : IEC_TMR
VERSION : 1.0
// stored: InstanceOfName IEC_TIMER
"IEC_TIMER"
BEGIN
END_DATA_BLOCK

DATA_BLOCK "IEC_Timer_6DB_1"   // DB38
{ S7_Optimized_Access := 'TRUE' }
AUTHOR : Simatic
FAMILY : IEC
NAME : IEC_TMR
VERSION : 1.0
// stored: InstanceOfName IEC_TIMER
"IEC_TIMER"
BEGIN
END_DATA_BLOCK

DATA_BLOCK "IEC_Timer_6DB_2"   // DB39
{ S7_Optimized_Access := 'TRUE' }
AUTHOR : Simatic
FAMILY : IEC
NAME : IEC_TMR
VERSION : 1.0
// stored: InstanceOfName IEC_TIMER
"IEC_TIMER"
BEGIN
END_DATA_BLOCK

DATA_BLOCK "IEC_Timer_6DB_3"   // DB40
{ S7_Optimized_Access := 'TRUE' }
AUTHOR : Simatic
FAMILY : IEC
NAME : IEC_TMR
VERSION : 1.0
// stored: InstanceOfName IEC_TIMER
"IEC_TIMER"
BEGIN
END_DATA_BLOCK

DATA_BLOCK "IEC_Timer_6DB_4"   // DB41
{ S7_Optimized_Access := 'TRUE' }
AUTHOR : Simatic
FAMILY : IEC
NAME : IEC_TMR
VERSION : 1.0
// stored: InstanceOfName IEC_TIMER
"IEC_TIMER"
BEGIN
END_DATA_BLOCK

DATA_BLOCK "IEC_Timer_6DB_5"   // DB42
{ S7_Optimized_Access := 'TRUE' }
AUTHOR : Simatic
FAMILY : IEC
NAME : IEC_TMR
VERSION : 1.0
// stored: InstanceOfName IEC_TIMER
"IEC_TIMER"
BEGIN
END_DATA_BLOCK

DATA_BLOCK "IEC_Timer_6DB_6"   // DB43
{ S7_Optimized_Access := 'TRUE' }
AUTHOR : Simatic
FAMILY : IEC
NAME : IEC_TMR
VERSION : 1.0
// stored: InstanceOfName IEC_TIMER
"IEC_TIMER"
BEGIN
END_DATA_BLOCK

DATA_BLOCK "IEC_Timer_6DB_7"   // DB44
{ S7_Optimized_Access := 'TRUE' }
AUTHOR : Simatic
FAMILY : IEC
NAME : IEC_TMR
VERSION : 1.0
// stored: InstanceOfName IEC_TIMER
"IEC_TIMER"
BEGIN
END_DATA_BLOCK

DATA_BLOCK "IEC_Timer_6DB_8"   // DB45
{ S7_Optimized_Access := 'TRUE' }
AUTHOR : Simatic
FAMILY : IEC
NAME : IEC_TMR
VERSION : 1.0
// stored: InstanceOfName IEC_TIMER
"IEC_TIMER"
BEGIN
END_DATA_BLOCK

DATA_BLOCK "IEC_Timer_6DB_9"   // DB46
{ S7_Optimized_Access := 'TRUE' }
AUTHOR : Simatic
FAMILY : IEC
NAME : IEC_TMR
VERSION : 1.0
// stored: InstanceOfName IEC_TIMER
"IEC_TIMER"
BEGIN
END_DATA_BLOCK

DATA_BLOCK "IEC_Timer_6DB_10"   // DB47
{ S7_Optimized_Access := 'TRUE' }
AUTHOR : Simatic
FAMILY : IEC
NAME : IEC_TMR
VERSION : 1.0
// stored: InstanceOfName IEC_TIMER
"IEC_TIMER"
BEGIN
END_DATA_BLOCK

DATA_BLOCK "IEC_Timer_6DB_12"   // DB48
{ S7_Optimized_Access := 'TRUE' }
AUTHOR : Simatic
FAMILY : IEC
NAME : IEC_TMR
VERSION : 1.0
// stored: InstanceOfName IEC_TIMER
"IEC_TIMER"
BEGIN
END_DATA_BLOCK

DATA_BLOCK "IEC_Timer_6DB_13"   // DB49
{ S7_Optimized_Access := 'TRUE' }
AUTHOR : Simatic
FAMILY : IEC
NAME : IEC_TMR
VERSION : 1.0
// stored: InstanceOfName IEC_TIMER
"IEC_TIMER"
BEGIN
END_DATA_BLOCK

DATA_BLOCK "IEC_Timer_6DB_14"   // DB50
{ S7_Optimized_Access := 'TRUE' }
AUTHOR : Simatic
FAMILY : IEC
NAME : IEC_TMR
VERSION : 1.0
// stored: InstanceOfName IEC_TIMER
"IEC_TIMER"
BEGIN
END_DATA_BLOCK

DATA_BLOCK "IEC_Timer_6DB_15"   // DB51
{ S7_Optimized_Access := 'TRUE' }
AUTHOR : Simatic
FAMILY : IEC
NAME : IEC_TMR
VERSION : 1.0
// stored: InstanceOfName IEC_TIMER
"IEC_TIMER"
BEGIN
END_DATA_BLOCK

DATA_BLOCK "IEC_Timer_6DB_16"   // DB52
{ S7_Optimized_Access := 'TRUE' }
AUTHOR : Simatic
FAMILY : IEC
NAME : IEC_TMR
VERSION : 1.0
// stored: InstanceOfName IEC_TIMER
"IEC_TIMER"
BEGIN
END_DATA_BLOCK

DATA_BLOCK "IEC_Timer_6DB_17"   // DB53
{ S7_Optimized_Access := 'TRUE' }
AUTHOR : Simatic
FAMILY : IEC
NAME : IEC_TMR
VERSION : 1.0
// stored: InstanceOfName IEC_TIMER
"IEC_TIMER"
BEGIN
END_DATA_BLOCK

DATA_BLOCK "IEC_Timer_6DB_18"   // DB54
{ S7_Optimized_Access := 'TRUE' }
AUTHOR : Simatic
FAMILY : IEC
NAME : IEC_TMR
VERSION : 1.0
// stored: InstanceOfName IEC_TIMER
"IEC_TIMER"
BEGIN
END_DATA_BLOCK

// folder: (top level)

FUNCTION_BLOCK "fb_modbus通讯"   // FB2, LAD
{ S7_Optimized_Access := 'TRUE' }
VERSION : 0.1
BEGIN

REGION Network 1
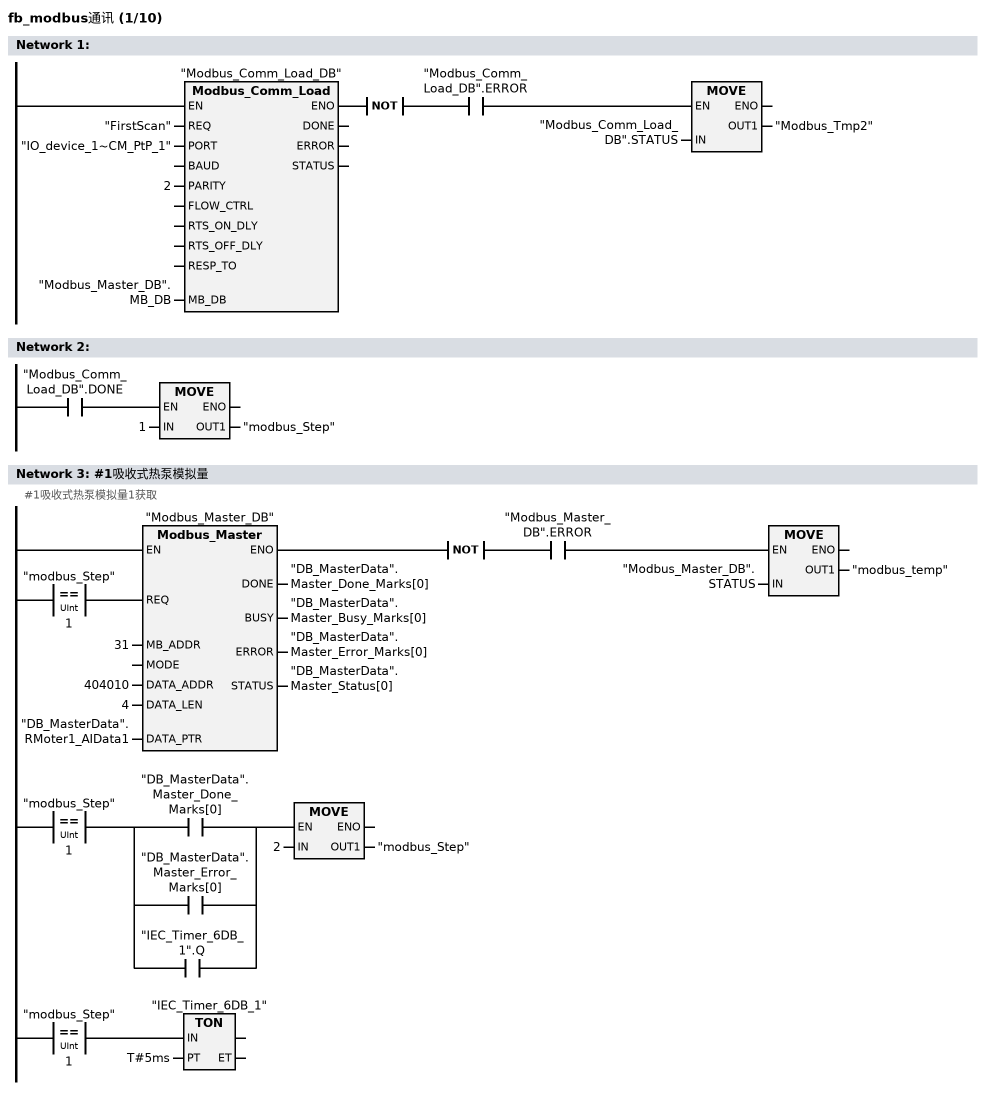
   // ENO of a box is taken as its EN; it also drops when the box reports an error
   "Modbus_Comm_Load_DB"(REQ := "FirstScan",   // Modbus_Comm_Load
                         PORT := "IO_device_1~CM_PtP_1",
                         PARITY := 2,
                         MB_DB := "Modbus_Master_DB".MB_DB);
   IF NOT TRUE AND "Modbus_Comm_Load_DB".ERROR THEN "Modbus_Tmp2" := "Modbus_Comm_Load_DB".STATUS; END_IF;
END_REGION

REGION Network 2
   RUNG wire#powerrail
      Contact( "Modbus_Comm_Load_DB".DONE )
      Move(in := 1, out1 => "modbus_Step")
   END_RUNG
   // the same network as SCL:
   IF "Modbus_Comm_Load_DB".DONE THEN "modbus_Step" := 1; END_IF;
END_REGION

REGION Network 3: #1吸收式热泵模拟量
   // #1吸收式热泵模拟量1获取
   // ENO of a box is taken as its EN; it also drops when the box reports an error
   "Modbus_Master_DB"(REQ := "modbus_Step" = 1,   // Modbus_Master
                      MB_ADDR := 31,
                      DATA_ADDR := 404010,
                      DATA_LEN := 4,
                      DATA_PTR := "DB_MasterData".RMoter1_AIData1,
                      DONE => "DB_MasterData".Master_Done_Marks[0],
                      BUSY => "DB_MasterData".Master_Busy_Marks[0],
                      ERROR => "DB_MasterData".Master_Error_Marks[0],
                      STATUS => "DB_MasterData".Master_Status[0]);
   IF NOT TRUE AND "Modbus_Master_DB".ERROR THEN "modbus_temp" := "Modbus_Master_DB".STATUS; END_IF;
   IF ("modbus_Step" = 1) AND ("DB_MasterData".Master_Done_Marks[0] OR "DB_MasterData".Master_Error_Marks[0] OR "IEC_Timer_6DB_1".Q) THEN
       "modbus_Step" := 2;
   END_IF;
   "IEC_Timer_6DB_1".TON(IN := "modbus_Step" = 1, PT := T#5ms);
END_REGION

REGION Network 4
   // #1吸收式热泵模拟量2获取
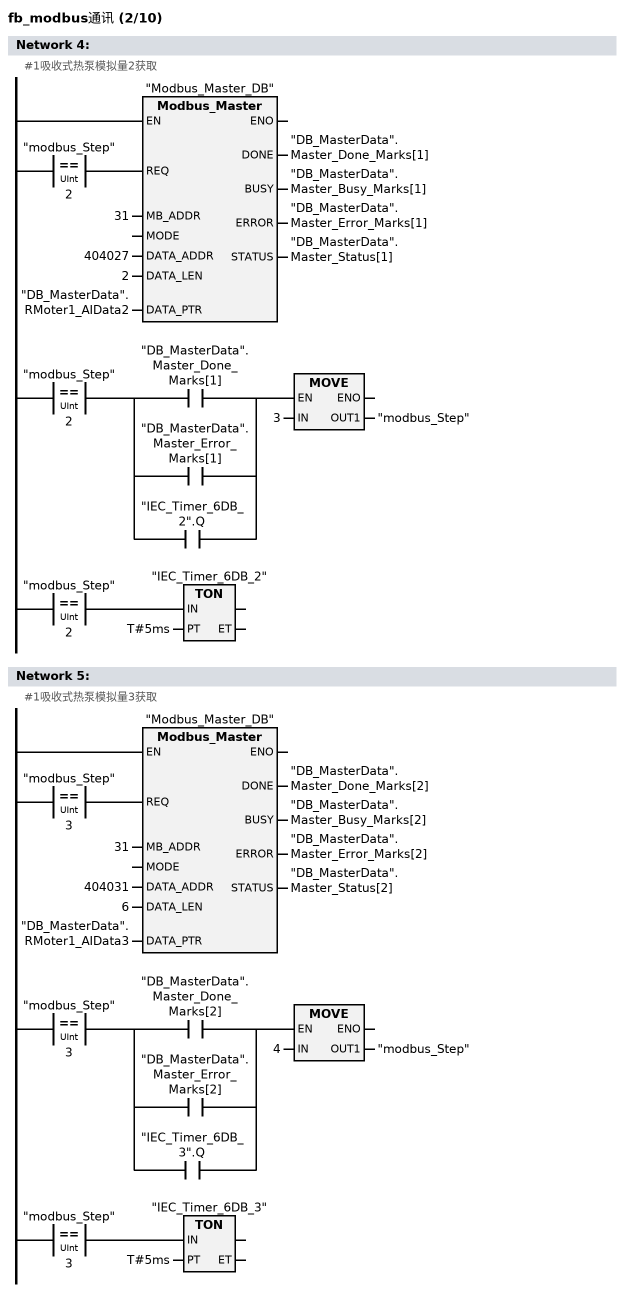
   "Modbus_Master_DB"(REQ := "modbus_Step" = 2,   // Modbus_Master
                      MB_ADDR := 31,
                      DATA_ADDR := 404027,
                      DATA_LEN := 2,
                      DATA_PTR := "DB_MasterData".RMoter1_AIData2,
                      DONE => "DB_MasterData".Master_Done_Marks[1],
                      BUSY => "DB_MasterData".Master_Busy_Marks[1],
                      ERROR => "DB_MasterData".Master_Error_Marks[1],
                      STATUS => "DB_MasterData".Master_Status[1]);
   IF ("modbus_Step" = 2) AND ("DB_MasterData".Master_Done_Marks[1] OR "DB_MasterData".Master_Error_Marks[1] OR "IEC_Timer_6DB_2".Q) THEN
       "modbus_Step" := 3;
   END_IF;
   "IEC_Timer_6DB_2".TON(IN := "modbus_Step" = 2, PT := T#5ms);
END_REGION

REGION Network 5
   // #1吸收式热泵模拟量3获取
   "Modbus_Master_DB"(REQ := "modbus_Step" = 3,   // Modbus_Master
                      MB_ADDR := 31,
                      DATA_ADDR := 404031,
                      DATA_LEN := 6,
                      DATA_PTR := "DB_MasterData".RMoter1_AIData3,
                      DONE => "DB_MasterData".Master_Done_Marks[2],
                      BUSY => "DB_MasterData".Master_Busy_Marks[2],
                      ERROR => "DB_MasterData".Master_Error_Marks[2],
                      STATUS => "DB_MasterData".Master_Status[2]);
   IF ("modbus_Step" = 3) AND ("DB_MasterData".Master_Done_Marks[2] OR "DB_MasterData".Master_Error_Marks[2] OR "IEC_Timer_6DB_3".Q) THEN
       "modbus_Step" := 4;
   END_IF;
   "IEC_Timer_6DB_3".TON(IN := "modbus_Step" = 3, PT := T#5ms);
END_REGION

REGION Network 6
   // #1吸收式热泵状态获取
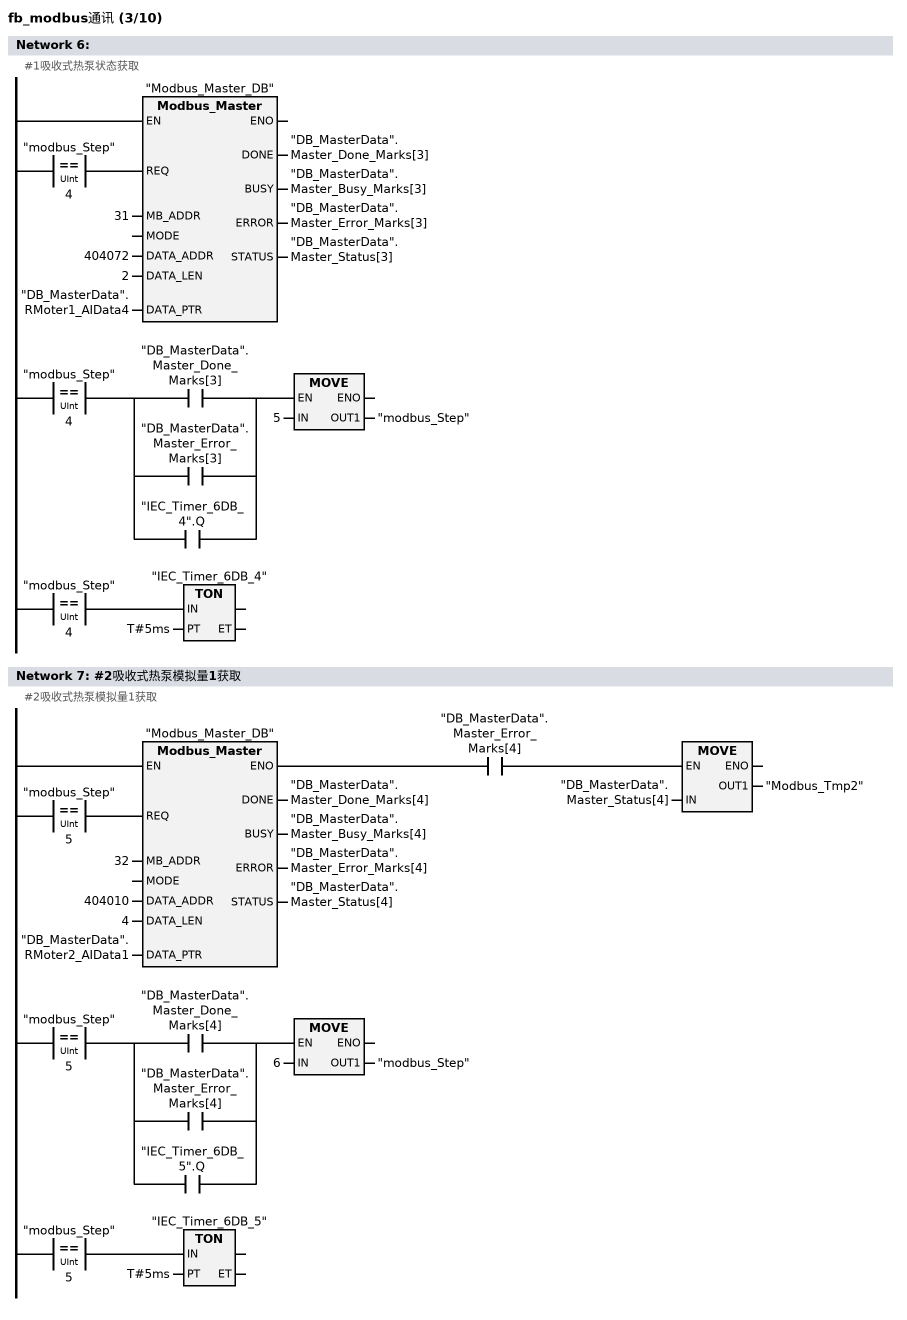
   "Modbus_Master_DB"(REQ := "modbus_Step" = 4,   // Modbus_Master
                      MB_ADDR := 31,
                      DATA_ADDR := 404072,
                      DATA_LEN := 2,
                      DATA_PTR := "DB_MasterData".RMoter1_AIData4,
                      DONE => "DB_MasterData".Master_Done_Marks[3],
                      BUSY => "DB_MasterData".Master_Busy_Marks[3],
                      ERROR => "DB_MasterData".Master_Error_Marks[3],
                      STATUS => "DB_MasterData".Master_Status[3]);
   IF ("modbus_Step" = 4) AND ("DB_MasterData".Master_Done_Marks[3] OR "DB_MasterData".Master_Error_Marks[3] OR "IEC_Timer_6DB_4".Q) THEN
       "modbus_Step" := 5;
   END_IF;
   "IEC_Timer_6DB_4".TON(IN := "modbus_Step" = 4, PT := T#5ms);
END_REGION

REGION Network 7: #2吸收式热泵模拟量1获取
   // #2吸收式热泵模拟量1获取
   // ENO of a box is taken as its EN; it also drops when the box reports an error
   "Modbus_Master_DB"(REQ := "modbus_Step" = 5,   // Modbus_Master
                      MB_ADDR := 32,
                      DATA_ADDR := 404010,
                      DATA_LEN := 4,
                      DATA_PTR := "DB_MasterData".RMoter2_AIData1,
                      DONE => "DB_MasterData".Master_Done_Marks[4],
                      BUSY => "DB_MasterData".Master_Busy_Marks[4],
                      ERROR => "DB_MasterData".Master_Error_Marks[4],
                      STATUS => "DB_MasterData".Master_Status[4]);
   IF "DB_MasterData".Master_Error_Marks[4] THEN "Modbus_Tmp2" := "DB_MasterData".Master_Status[4]; END_IF;
   IF ("modbus_Step" = 5) AND ("DB_MasterData".Master_Done_Marks[4] OR "DB_MasterData".Master_Error_Marks[4] OR "IEC_Timer_6DB_5".Q) THEN
       "modbus_Step" := 6;
   END_IF;
   "IEC_Timer_6DB_5".TON(IN := "modbus_Step" = 5, PT := T#5ms);
END_REGION

REGION Network 8
   // #1吸收式热泵模拟量2获取
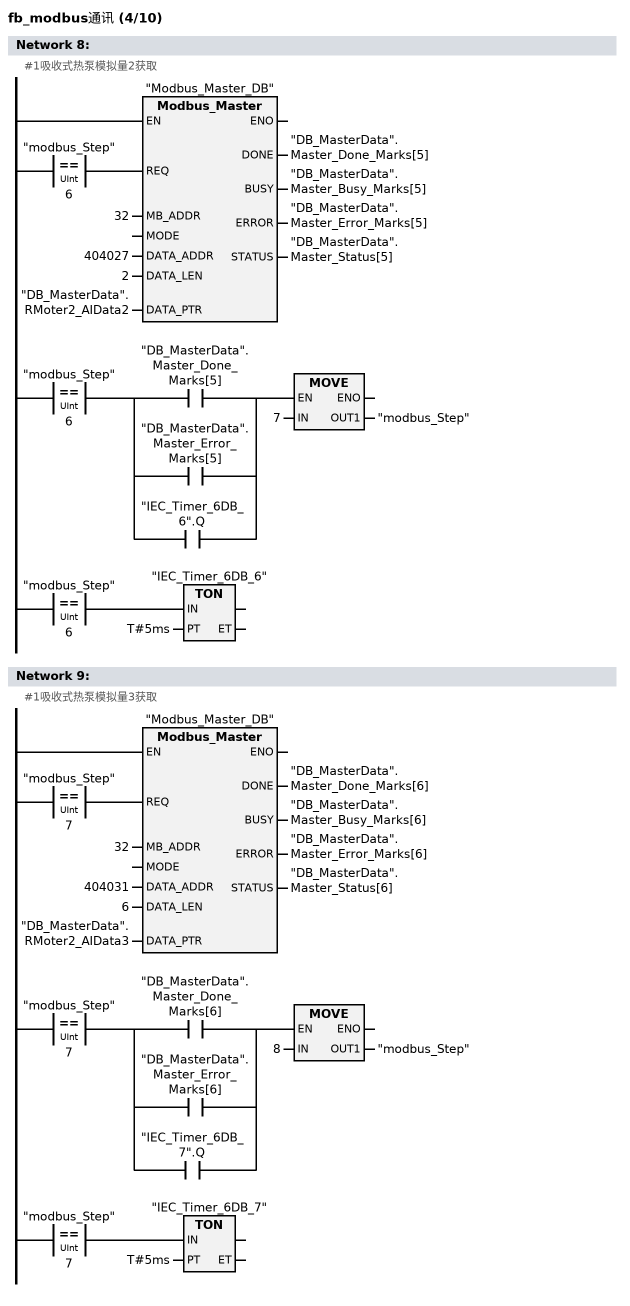
   "Modbus_Master_DB"(REQ := "modbus_Step" = 6,   // Modbus_Master
                      MB_ADDR := 32,
                      DATA_ADDR := 404027,
                      DATA_LEN := 2,
                      DATA_PTR := "DB_MasterData".RMoter2_AIData2,
                      DONE => "DB_MasterData".Master_Done_Marks[5],
                      BUSY => "DB_MasterData".Master_Busy_Marks[5],
                      ERROR => "DB_MasterData".Master_Error_Marks[5],
                      STATUS => "DB_MasterData".Master_Status[5]);
   IF ("modbus_Step" = 6) AND ("DB_MasterData".Master_Done_Marks[5] OR "DB_MasterData".Master_Error_Marks[5] OR "IEC_Timer_6DB_6".Q) THEN
       "modbus_Step" := 7;
   END_IF;
   "IEC_Timer_6DB_6".TON(IN := "modbus_Step" = 6, PT := T#5ms);
END_REGION

REGION Network 9
   // #1吸收式热泵模拟量3获取
   "Modbus_Master_DB"(REQ := "modbus_Step" = 7,   // Modbus_Master
                      MB_ADDR := 32,
                      DATA_ADDR := 404031,
                      DATA_LEN := 6,
                      DATA_PTR := "DB_MasterData".RMoter2_AIData3,
                      DONE => "DB_MasterData".Master_Done_Marks[6],
                      BUSY => "DB_MasterData".Master_Busy_Marks[6],
                      ERROR => "DB_MasterData".Master_Error_Marks[6],
                      STATUS => "DB_MasterData".Master_Status[6]);
   IF ("modbus_Step" = 7) AND ("DB_MasterData".Master_Done_Marks[6] OR "DB_MasterData".Master_Error_Marks[6] OR "IEC_Timer_6DB_7".Q) THEN
       "modbus_Step" := 8;
   END_IF;
   "IEC_Timer_6DB_7".TON(IN := "modbus_Step" = 7, PT := T#5ms);
END_REGION

REGION Network 10
   // #1吸收式热泵状态获取
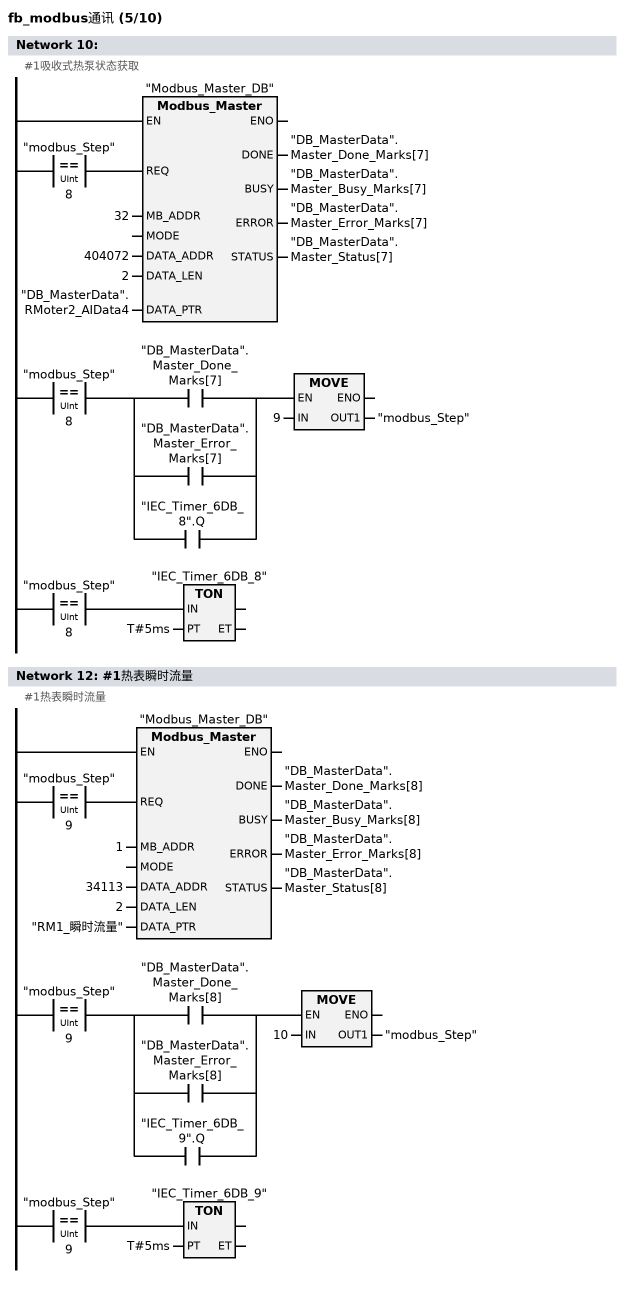
   "Modbus_Master_DB"(REQ := "modbus_Step" = 8,   // Modbus_Master
                      MB_ADDR := 32,
                      DATA_ADDR := 404072,
                      DATA_LEN := 2,
                      DATA_PTR := "DB_MasterData".RMoter2_AIData4,
                      DONE => "DB_MasterData".Master_Done_Marks[7],
                      BUSY => "DB_MasterData".Master_Busy_Marks[7],
                      ERROR => "DB_MasterData".Master_Error_Marks[7],
                      STATUS => "DB_MasterData".Master_Status[7]);
   IF ("modbus_Step" = 8) AND ("DB_MasterData".Master_Done_Marks[7] OR "DB_MasterData".Master_Error_Marks[7] OR "IEC_Timer_6DB_8".Q) THEN
       "modbus_Step" := 9;
   END_IF;
   "IEC_Timer_6DB_8".TON(IN := "modbus_Step" = 8, PT := T#5ms);
END_REGION

REGION Network 12: #1热表瞬时流量
   // #1热表瞬时流量
   "Modbus_Master_DB"(REQ := "modbus_Step" = 9,   // Modbus_Master
                      MB_ADDR := 1,
                      DATA_ADDR := 34113,
                      DATA_LEN := 2,
                      DATA_PTR := "RM1_瞬时流量",
                      DONE => "DB_MasterData".Master_Done_Marks[8],
                      BUSY => "DB_MasterData".Master_Busy_Marks[8],
                      ERROR => "DB_MasterData".Master_Error_Marks[8],
                      STATUS => "DB_MasterData".Master_Status[8]);
   IF ("modbus_Step" = 9) AND ("DB_MasterData".Master_Done_Marks[8] OR "DB_MasterData".Master_Error_Marks[8] OR "IEC_Timer_6DB_9".Q) THEN
       "modbus_Step" := 10;
   END_IF;
   "IEC_Timer_6DB_9".TON(IN := "modbus_Step" = 9, PT := T#5ms);
END_REGION

REGION Network 13: #1热表瞬时热量、累计热量、出入口温度
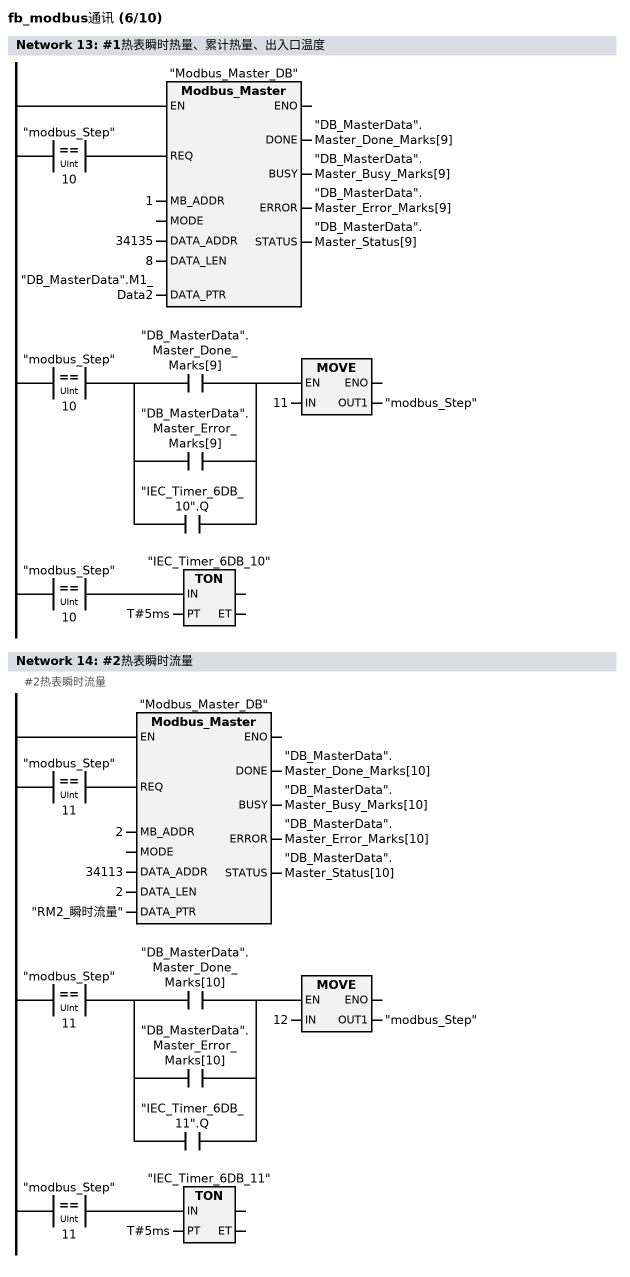
   "Modbus_Master_DB"(REQ := "modbus_Step" = 10,   // Modbus_Master
                      MB_ADDR := 1,
                      DATA_ADDR := 34135,
                      DATA_LEN := 8,
                      DATA_PTR := "DB_MasterData".M1_Data2,
                      DONE => "DB_MasterData".Master_Done_Marks[9],
                      BUSY => "DB_MasterData".Master_Busy_Marks[9],
                      ERROR => "DB_MasterData".Master_Error_Marks[9],
                      STATUS => "DB_MasterData".Master_Status[9]);
   IF ("modbus_Step" = 10) AND ("DB_MasterData".Master_Done_Marks[9] OR "DB_MasterData".Master_Error_Marks[9] OR "IEC_Timer_6DB_10".Q) THEN
       "modbus_Step" := 11;
   END_IF;
   "IEC_Timer_6DB_10".TON(IN := "modbus_Step" = 10, PT := T#5ms);
END_REGION

REGION Network 14: #2热表瞬时流量
   // #2热表瞬时流量
   "Modbus_Master_DB"(REQ := "modbus_Step" = 11,   // Modbus_Master
                      MB_ADDR := 2,
                      DATA_ADDR := 34113,
                      DATA_LEN := 2,
                      DATA_PTR := "RM2_瞬时流量",
                      DONE => "DB_MasterData".Master_Done_Marks[10],
                      BUSY => "DB_MasterData".Master_Busy_Marks[10],
                      ERROR => "DB_MasterData".Master_Error_Marks[10],
                      STATUS => "DB_MasterData".Master_Status[10]);
   IF ("modbus_Step" = 11) AND ("DB_MasterData".Master_Done_Marks[10] OR "DB_MasterData".Master_Error_Marks[10] OR "IEC_Timer_6DB_11".Q) THEN
       "modbus_Step" := 12;
   END_IF;
   "IEC_Timer_6DB_11".TON(IN := "modbus_Step" = 11, PT := T#5ms);
END_REGION

REGION Network 15: #2热表瞬时热量、累计热量、出入口温度
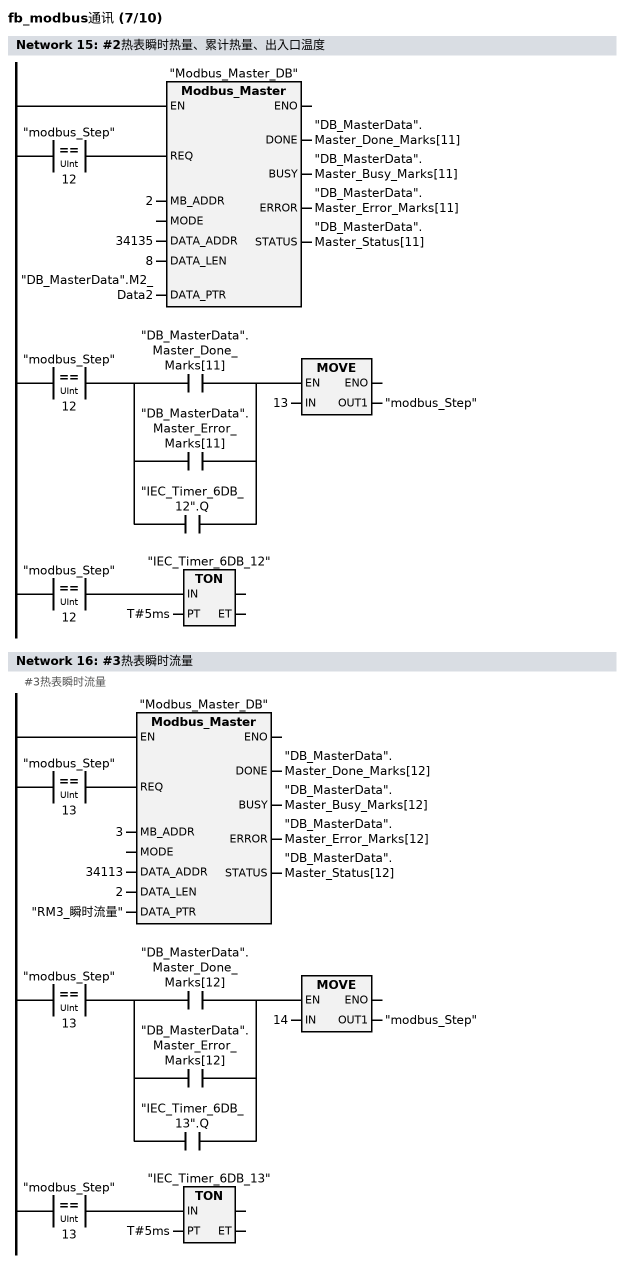
   "Modbus_Master_DB"(REQ := "modbus_Step" = 12,   // Modbus_Master
                      MB_ADDR := 2,
                      DATA_ADDR := 34135,
                      DATA_LEN := 8,
                      DATA_PTR := "DB_MasterData".M2_Data2,
                      DONE => "DB_MasterData".Master_Done_Marks[11],
                      BUSY => "DB_MasterData".Master_Busy_Marks[11],
                      ERROR => "DB_MasterData".Master_Error_Marks[11],
                      STATUS => "DB_MasterData".Master_Status[11]);
   IF ("modbus_Step" = 12) AND ("DB_MasterData".Master_Done_Marks[11] OR "DB_MasterData".Master_Error_Marks[11] OR "IEC_Timer_6DB_12".Q) THEN
       "modbus_Step" := 13;
   END_IF;
   "IEC_Timer_6DB_12".TON(IN := "modbus_Step" = 12, PT := T#5ms);
END_REGION

REGION Network 16: #3热表瞬时流量
   // #3热表瞬时流量
   "Modbus_Master_DB"(REQ := "modbus_Step" = 13,   // Modbus_Master
                      MB_ADDR := 3,
                      DATA_ADDR := 34113,
                      DATA_LEN := 2,
                      DATA_PTR := "RM3_瞬时流量",
                      DONE => "DB_MasterData".Master_Done_Marks[12],
                      BUSY => "DB_MasterData".Master_Busy_Marks[12],
                      ERROR => "DB_MasterData".Master_Error_Marks[12],
                      STATUS => "DB_MasterData".Master_Status[12]);
   IF ("modbus_Step" = 13) AND ("DB_MasterData".Master_Done_Marks[12] OR "DB_MasterData".Master_Error_Marks[12] OR "IEC_Timer_6DB_13".Q) THEN
       "modbus_Step" := 14;
   END_IF;
   "IEC_Timer_6DB_13".TON(IN := "modbus_Step" = 13, PT := T#5ms);
END_REGION

REGION Network 17: #3热表瞬时热量、累计热量、出入口温度
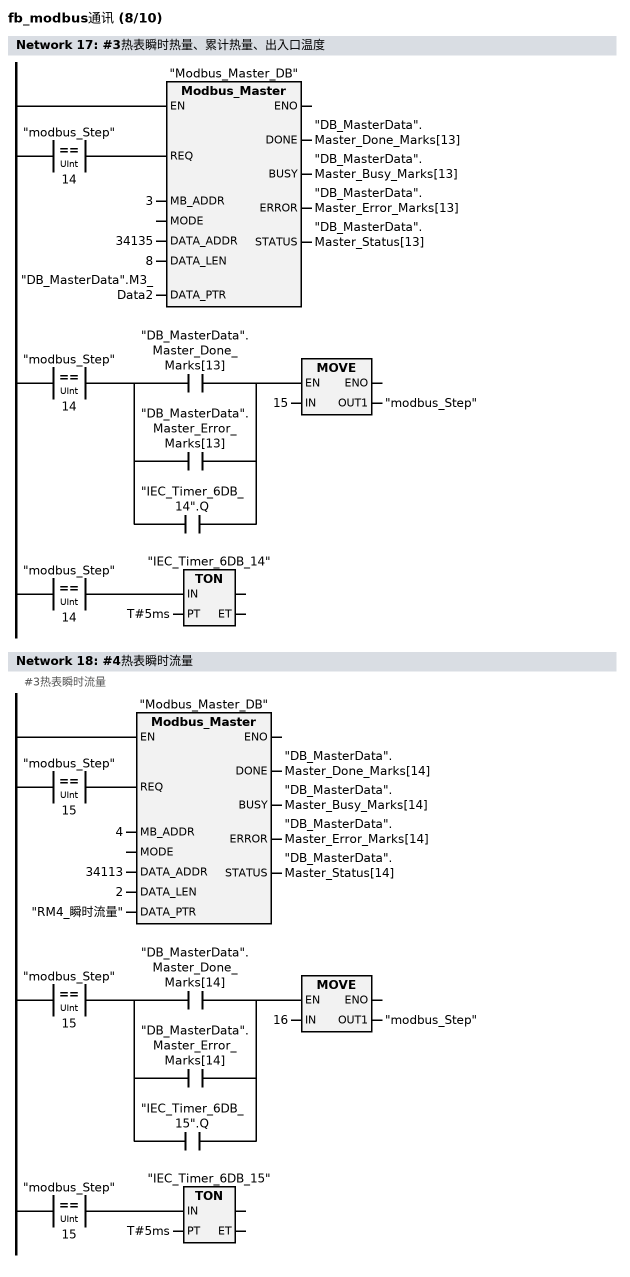
   "Modbus_Master_DB"(REQ := "modbus_Step" = 14,   // Modbus_Master
                      MB_ADDR := 3,
                      DATA_ADDR := 34135,
                      DATA_LEN := 8,
                      DATA_PTR := "DB_MasterData".M3_Data2,
                      DONE => "DB_MasterData".Master_Done_Marks[13],
                      BUSY => "DB_MasterData".Master_Busy_Marks[13],
                      ERROR => "DB_MasterData".Master_Error_Marks[13],
                      STATUS => "DB_MasterData".Master_Status[13]);
   IF ("modbus_Step" = 14) AND ("DB_MasterData".Master_Done_Marks[13] OR "DB_MasterData".Master_Error_Marks[13] OR "IEC_Timer_6DB_14".Q) THEN
       "modbus_Step" := 15;
   END_IF;
   "IEC_Timer_6DB_14".TON(IN := "modbus_Step" = 14, PT := T#5ms);
END_REGION

REGION Network 18: #4热表瞬时流量
   // #3热表瞬时流量
   "Modbus_Master_DB"(REQ := "modbus_Step" = 15,   // Modbus_Master
                      MB_ADDR := 4,
                      DATA_ADDR := 34113,
                      DATA_LEN := 2,
                      DATA_PTR := "RM4_瞬时流量",
                      DONE => "DB_MasterData".Master_Done_Marks[14],
                      BUSY => "DB_MasterData".Master_Busy_Marks[14],
                      ERROR => "DB_MasterData".Master_Error_Marks[14],
                      STATUS => "DB_MasterData".Master_Status[14]);
   IF ("modbus_Step" = 15) AND ("DB_MasterData".Master_Done_Marks[14] OR "DB_MasterData".Master_Error_Marks[14] OR "IEC_Timer_6DB_15".Q) THEN
       "modbus_Step" := 16;
   END_IF;
   "IEC_Timer_6DB_15".TON(IN := "modbus_Step" = 15, PT := T#5ms);
END_REGION

REGION Network 19: #4热表瞬时热量、累计热量、出入口温度
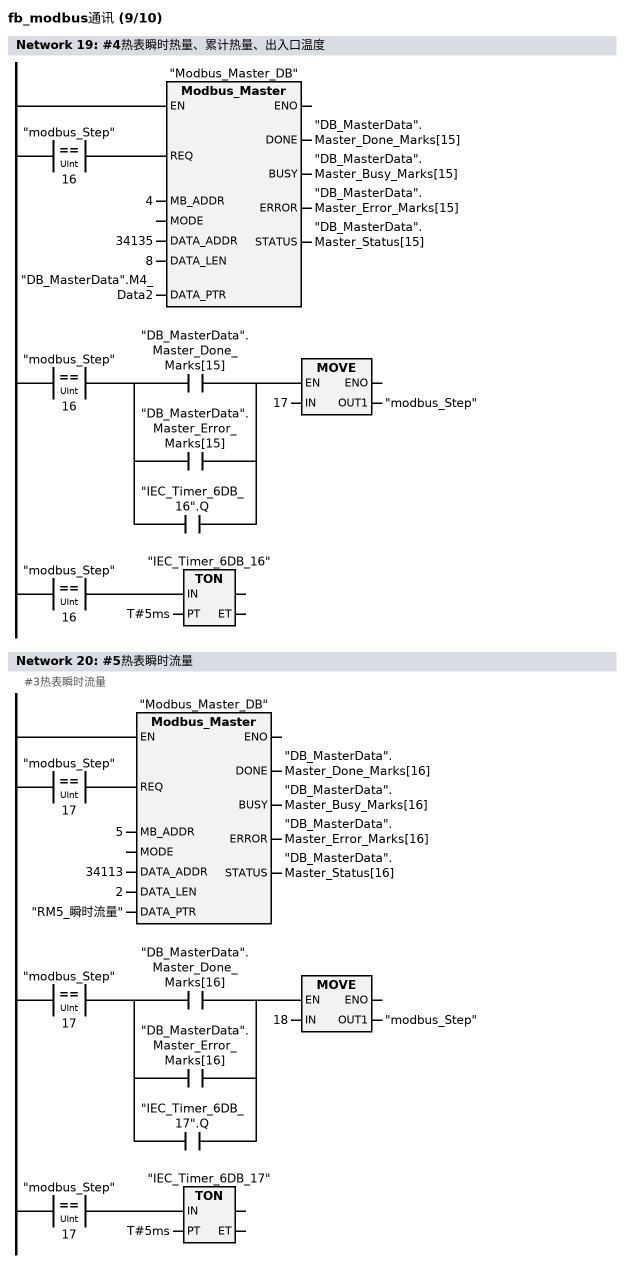
   "Modbus_Master_DB"(REQ := "modbus_Step" = 16,   // Modbus_Master
                      MB_ADDR := 4,
                      DATA_ADDR := 34135,
                      DATA_LEN := 8,
                      DATA_PTR := "DB_MasterData".M4_Data2,
                      DONE => "DB_MasterData".Master_Done_Marks[15],
                      BUSY => "DB_MasterData".Master_Busy_Marks[15],
                      ERROR => "DB_MasterData".Master_Error_Marks[15],
                      STATUS => "DB_MasterData".Master_Status[15]);
   IF ("modbus_Step" = 16) AND ("DB_MasterData".Master_Done_Marks[15] OR "DB_MasterData".Master_Error_Marks[15] OR "IEC_Timer_6DB_16".Q) THEN
       "modbus_Step" := 17;
   END_IF;
   "IEC_Timer_6DB_16".TON(IN := "modbus_Step" = 16, PT := T#5ms);
END_REGION

REGION Network 20: #5热表瞬时流量
   // #3热表瞬时流量
   "Modbus_Master_DB"(REQ := "modbus_Step" = 17,   // Modbus_Master
                      MB_ADDR := 5,
                      DATA_ADDR := 34113,
                      DATA_LEN := 2,
                      DATA_PTR := "RM5_瞬时流量",
                      DONE => "DB_MasterData".Master_Done_Marks[16],
                      BUSY => "DB_MasterData".Master_Busy_Marks[16],
                      ERROR => "DB_MasterData".Master_Error_Marks[16],
                      STATUS => "DB_MasterData".Master_Status[16]);
   IF ("modbus_Step" = 17) AND ("DB_MasterData".Master_Done_Marks[16] OR "DB_MasterData".Master_Error_Marks[16] OR "IEC_Timer_6DB_17".Q) THEN
       "modbus_Step" := 18;
   END_IF;
   "IEC_Timer_6DB_17".TON(IN := "modbus_Step" = 17, PT := T#5ms);
END_REGION

REGION Network 21: #5热表瞬时热量、累计热量、出入口温度
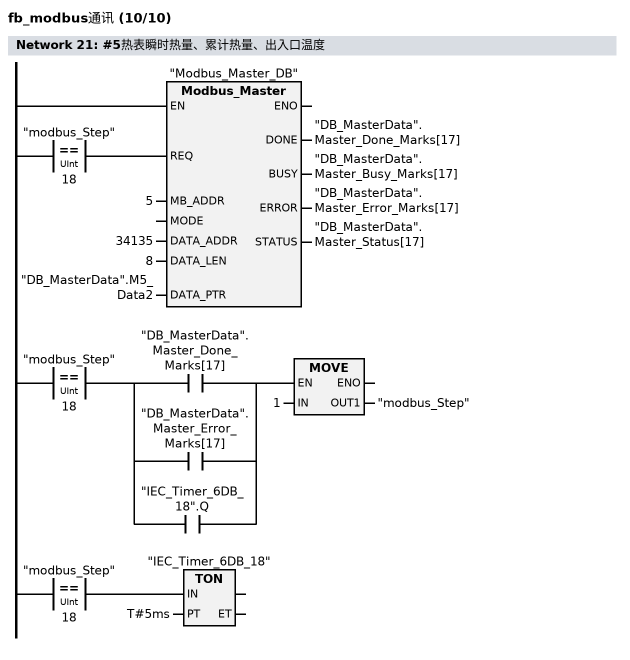
   "Modbus_Master_DB"(REQ := "modbus_Step" = 18,   // Modbus_Master
                      MB_ADDR := 5,
                      DATA_ADDR := 34135,
                      DATA_LEN := 8,
                      DATA_PTR := "DB_MasterData".M5_Data2,
                      DONE => "DB_MasterData".Master_Done_Marks[17],
                      BUSY => "DB_MasterData".Master_Busy_Marks[17],
                      ERROR => "DB_MasterData".Master_Error_Marks[17],
                      STATUS => "DB_MasterData".Master_Status[17]);
   IF ("modbus_Step" = 18) AND ("DB_MasterData".Master_Done_Marks[17] OR "DB_MasterData".Master_Error_Marks[17] OR "IEC_Timer_6DB_18".Q) THEN
       "modbus_Step" := 1;
   END_IF;
   "IEC_Timer_6DB_18".TON(IN := "modbus_Step" = 18, PT := T#5ms);
END_REGION
END_FUNCTION_BLOCK

FUNCTION "fc_模拟量转化" : Void   // FC1, LAD
{ S7_Optimized_Access := 'TRUE' }
VERSION : 0.1
   VAR_INPUT
      origin : Word;
      High : Real;
      Low : Real;
      Diff : Real;
   END_VAR
   VAR_OUTPUT
      CValue : Real;
      RVaule : Real;
   END_VAR
   VAR_TEMP
      Tmp1 : Real;
      Tmp2 : Real;
   END_VAR
BEGIN

REGION Network 1
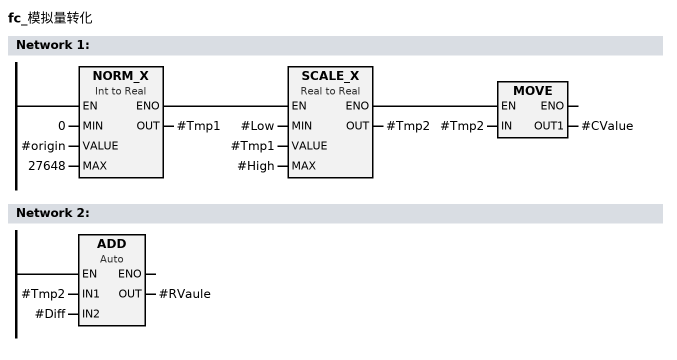
   RUNG wire#powerrail
      { S7_Templates := "[SrcType := Int, DestType := Real]" } Normalize(min := 0, value := #origin, max := 27648, out => #Tmp1)
      { S7_Templates := "[SrcType := Real, DestType := Real]" } Scale(min := #Low, value := #Tmp1, max := #High, out => #Tmp2)
      Move(in := #Tmp2, out1 => #CValue)
   END_RUNG
   // the same network as SCL:
   #Tmp1 := NORM_X(MIN := 0, VALUE := #origin, MAX := 27648);
   #Tmp2 := SCALE_X(MIN := #Low, VALUE := #Tmp1, MAX := #High);
   #CValue := #Tmp2;
END_REGION

REGION Network 2
   RUNG wire#powerrail
      Add(in1 := #Tmp2, in2 := #Diff, out => #RVaule)
   END_RUNG
   // the same network as SCL:
   #RVaule := #Tmp2 + #Diff;
END_REGION
END_FUNCTION

FUNCTION "cmp_array_bool" : Void   // FC2, SCL
{ S7_Optimized_Access := 'TRUE' }
VERSION : 0.1
   VAR_INPUT
      iArray : Array[0..32] of Bool;
   END_VAR
   VAR_OUTPUT
      result : Bool;
   END_VAR
   VAR_TEMP
      index : Int;
      value : Bool;
   END_VAR
BEGIN
       FOR #index := 0 TO 32 DO
           // Statement section FOR
           #result := #iArray[#index] = TRUE;
           IF #result THEN
               EXIT;// Statement section IF
           END_IF;
       END_FOR;
END_FUNCTION

FUNCTION "cmp_arrar_real" : Void   // FC3, SCL
{ S7_Optimized_Access := 'TRUE' }
VERSION : 0.1
// 比较上下限,报警
   VAR_INPUT
      inputSet : Array[0..1] of Real;
      inputValue : Real;
   END_VAR
   VAR_OUTPUT
      result : Bool;
   END_VAR
   VAR_TEMP
      index : Int;
      maxValue : Real;
      minValue : Real;
   END_VAR
BEGIN
   #maxValue := #inputSet[0];
   #minValue := #inputSet[1];

   IF #inputValue>#maxValue OR #inputValue<#minValue  THEN
       #result := TRUE;
   ELSE
       #result := FALSE;
       // Statement section IF
   END_IF;
END_FUNCTION

FUNCTION "fc_报警处理模块" : Void   // FC4, LAD
{ S7_Optimized_Access := 'TRUE' }
VERSION : 0.1
   VAR_INPUT
      Value : Real;
      Sets : Array[0..1] of Real;
      DelayT : DWord;
   END_VAR
   VAR_OUTPUT
      result : Bool;
   END_VAR
   VAR_TEMP
      _OK_ : Bool;
      _CuTm_ : DWord;
   END_VAR
BEGIN

REGION Network 1
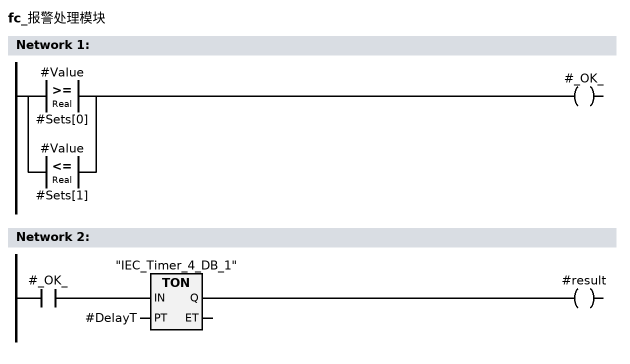
   RUNG wire#powerrail
      { S7_Templates := "SrcType := Real" } GE_Contact(in1 := #Value, in2 := #Sets[0])
      wire#w1
      Coil( #_OK_ )
   END_RUNG
   RUNG wire#powerrail
      { S7_Templates := "SrcType := Real" } LE_Contact(in1 := #Value, in2 := #Sets[1])
   END_RUNG wire#w1
   // the same network as SCL:
   #_OK_ := (#Value >= #Sets[0]) OR (#Value <= #Sets[1]);
END_REGION

REGION Network 2
   "IEC_Timer_4_DB_1".TON(IN := #_OK_, PT := #DelayT);
   #result := "IEC_Timer_4_DB_1".Q;
END_REGION
END_FUNCTION

ORGANIZATION_BLOCK "Main"   // OB1, LAD, ProgramCycle
TITLE = "Main Program Sweep (Cycle)"
{ S7_Optimized_Access := 'TRUE' }
VERSION : 0.1
   VAR_INPUT
      Initial_Call : Bool;   // Initial call of this OB
      Remanence : Bool;   // =True, if remanent data are available
   END_VAR
   VAR_TEMP   // added for the SCL form of the ladder/FBD networks
      _w1 : Bool;
   END_VAR
BEGIN

REGION Network 1
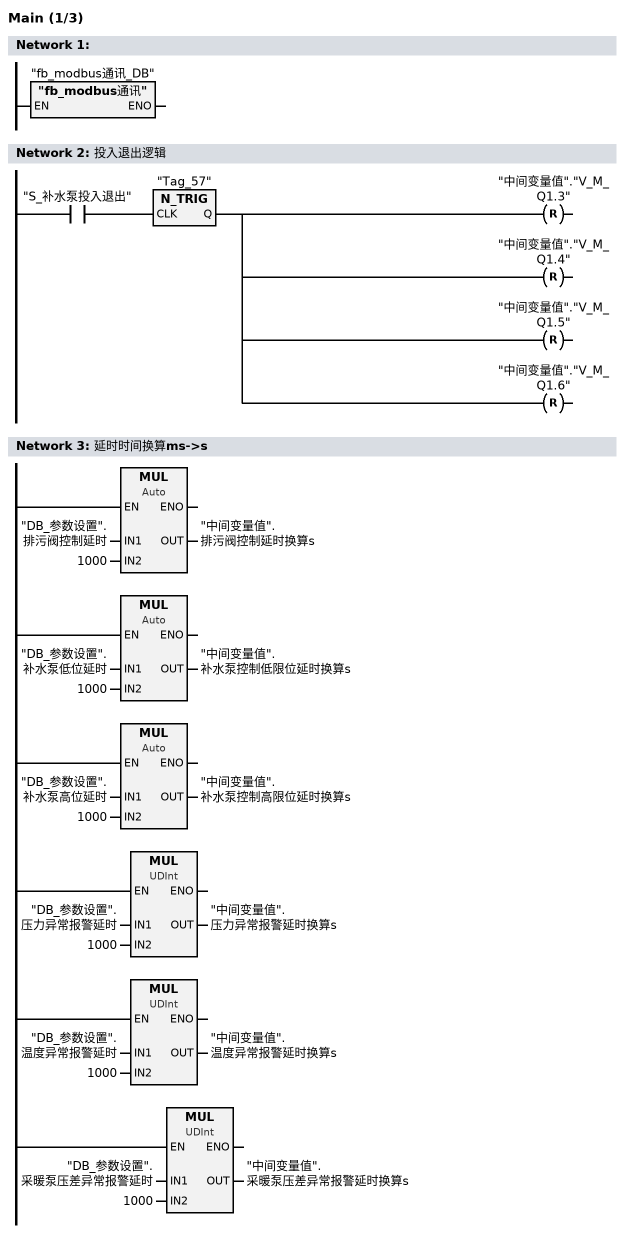
   RUNG wire#powerrail
      "fb_modbus通讯_DB"()
   END_RUNG
   // the same network as SCL:
   "fb_modbus通讯_DB"();   // "fb_modbus通讯"
END_REGION

REGION Network 2: 投入退出逻辑
   RUNG wire#powerrail
      Contact( "S_补水泵投入退出" )
      N_Trig( "Tag_57" )
      wire#w1
      R_Coil( "中间变量值"."V_M_Q1.3" )
   END_RUNG
   RUNG wire#w1
      R_Coil( "中间变量值"."V_M_Q1.4" )
   END_RUNG
   RUNG wire#w1
      R_Coil( "中间变量值"."V_M_Q1.5" )
   END_RUNG
   RUNG wire#w1
      R_Coil( "中间变量值"."V_M_Q1.6" )
   END_RUNG
   // the same network as SCL:
   #_w1 := NOT "S_补水泵投入退出" AND "Tag_57";   // falling edge
   "Tag_57" := "S_补水泵投入退出";
   IF #_w1 THEN
       "中间变量值"."V_M_Q1.3" := FALSE;
       "中间变量值"."V_M_Q1.4" := FALSE;
       "中间变量值"."V_M_Q1.5" := FALSE;
       "中间变量值"."V_M_Q1.6" := FALSE;
   END_IF;
END_REGION

REGION Network 3: 延时时间换算ms->s
   RUNG wire#powerrail
      Mul(in1 := "DB_参数设置".排污阀控制延时, in2 := 1000, out => "中间变量值".排污阀控制延时换算s)
   END_RUNG
   RUNG wire#powerrail
      Mul(in1 := "DB_参数设置".补水泵低位延时, in2 := 1000, out => "中间变量值".补水泵控制低限位延时换算s)
   END_RUNG
   RUNG wire#powerrail
      Mul(in1 := "DB_参数设置".补水泵高位延时, in2 := 1000, out => "中间变量值".补水泵控制高限位延时换算s)
   END_RUNG
   RUNG wire#powerrail
      { S7_Templates := "SrcType := UDInt" } Mul(in1 := "DB_参数设置".压力异常报警延时, in2 := 1000, out => "中间变量值".压力异常报警延时换算s)
   END_RUNG
   RUNG wire#powerrail
      { S7_Templates := "SrcType := UDInt" } Mul(in1 := "DB_参数设置".温度异常报警延时, in2 := 1000, out => "中间变量值".温度异常报警延时换算s)
   END_RUNG
   RUNG wire#powerrail
      { S7_Templates := "SrcType := UDInt" } Mul(in1 := "DB_参数设置".采暖泵压差异常报警延时, in2 := 1000, out => "中间变量值".采暖泵压差异常报警延时换算s)
   END_RUNG
   // the same network as SCL:
   "中间变量值".排污阀控制延时换算s := "DB_参数设置".排污阀控制延时 * 1000;
   "中间变量值".补水泵控制低限位延时换算s := "DB_参数设置".补水泵低位延时 * 1000;
   "中间变量值".补水泵控制高限位延时换算s := "DB_参数设置".补水泵高位延时 * 1000;
   "中间变量值".压力异常报警延时换算s := "DB_参数设置".压力异常报警延时 * 1000;
   "中间变量值".温度异常报警延时换算s := "DB_参数设置".温度异常报警延时 * 1000;
   "中间变量值".采暖泵压差异常报警延时换算s := "DB_参数设置".采暖泵压差异常报警延时 * 1000;
END_REGION

REGION Network 4: 二网水泵控制
   // 二网水泵控制
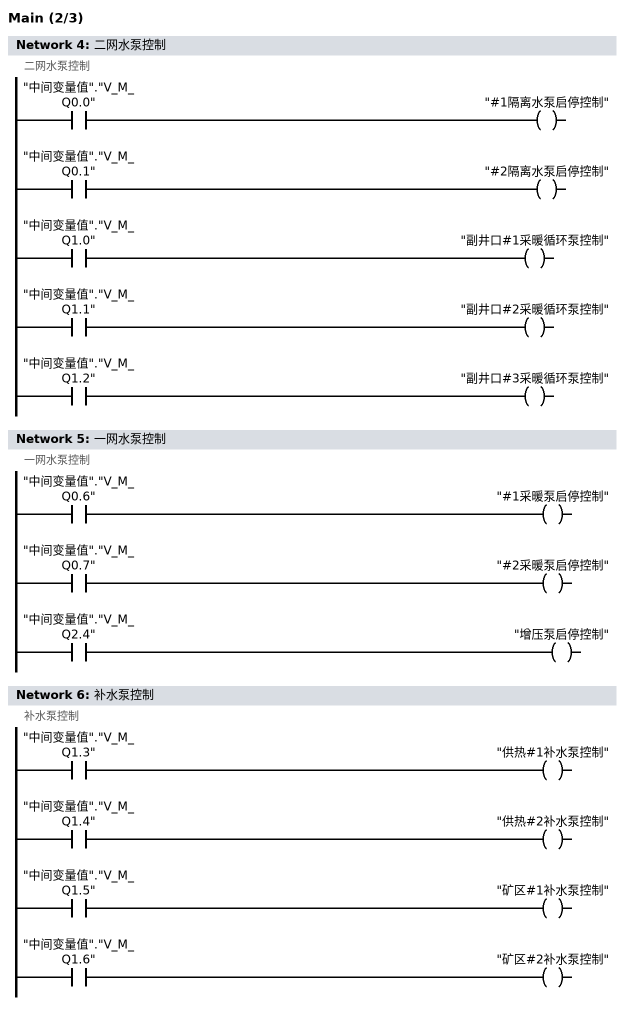
   RUNG wire#powerrail
      Contact( "中间变量值"."V_M_Q0.0" )
      Coil( "#1隔离水泵启停控制" )
   END_RUNG
   RUNG wire#powerrail
      Contact( "中间变量值"."V_M_Q0.1" )
      Coil( "#2隔离水泵启停控制" )
   END_RUNG
   RUNG wire#powerrail
      Contact( "中间变量值"."V_M_Q1.0" )
      Coil( "副井口#1采暖循环泵控制" )
   END_RUNG
   RUNG wire#powerrail
      Contact( "中间变量值"."V_M_Q1.1" )
      Coil( "副井口#2采暖循环泵控制" )
   END_RUNG
   RUNG wire#powerrail
      Contact( "中间变量值"."V_M_Q1.2" )
      Coil( "副井口#3采暖循环泵控制" )
   END_RUNG
   // the same network as SCL:
   "#1隔离水泵启停控制" := "中间变量值"."V_M_Q0.0";
   "#2隔离水泵启停控制" := "中间变量值"."V_M_Q0.1";
   "副井口#1采暖循环泵控制" := "中间变量值"."V_M_Q1.0";
   "副井口#2采暖循环泵控制" := "中间变量值"."V_M_Q1.1";
   "副井口#3采暖循环泵控制" := "中间变量值"."V_M_Q1.2";
END_REGION

REGION Network 5: 一网水泵控制
   // 一网水泵控制
   RUNG wire#powerrail
      Contact( "中间变量值"."V_M_Q0.6" )
      Coil( "#1采暖泵启停控制" )
   END_RUNG
   RUNG wire#powerrail
      Contact( "中间变量值"."V_M_Q0.7" )
      Coil( "#2采暖泵启停控制" )
   END_RUNG
   RUNG wire#powerrail
      Contact( "中间变量值"."V_M_Q2.4" )
      Coil( "增压泵启停控制" )
   END_RUNG
   // the same network as SCL:
   "#1采暖泵启停控制" := "中间变量值"."V_M_Q0.6";
   "#2采暖泵启停控制" := "中间变量值"."V_M_Q0.7";
   "增压泵启停控制" := "中间变量值"."V_M_Q2.4";
END_REGION

REGION Network 6: 补水泵控制
   // 补水泵控制
   RUNG wire#powerrail
      Contact( "中间变量值"."V_M_Q1.3" )
      Coil( "供热#1补水泵控制" )
   END_RUNG
   RUNG wire#powerrail
      Contact( "中间变量值"."V_M_Q1.4" )
      Coil( "供热#2补水泵控制" )
   END_RUNG
   RUNG wire#powerrail
      Contact( "中间变量值"."V_M_Q1.5" )
      Coil( "矿区#1补水泵控制" )
   END_RUNG
   RUNG wire#powerrail
      Contact( "中间变量值"."V_M_Q1.6" )
      Coil( "矿区#2补水泵控制" )
   END_RUNG
   // the same network as SCL:
   "供热#1补水泵控制" := "中间变量值"."V_M_Q1.3";
   "供热#2补水泵控制" := "中间变量值"."V_M_Q1.4";
   "矿区#1补水泵控制" := "中间变量值"."V_M_Q1.5";
   "矿区#2补水泵控制" := "中间变量值"."V_M_Q1.6";
END_REGION

REGION Network 7: 电磁阀控制
   // 电磁阀控制
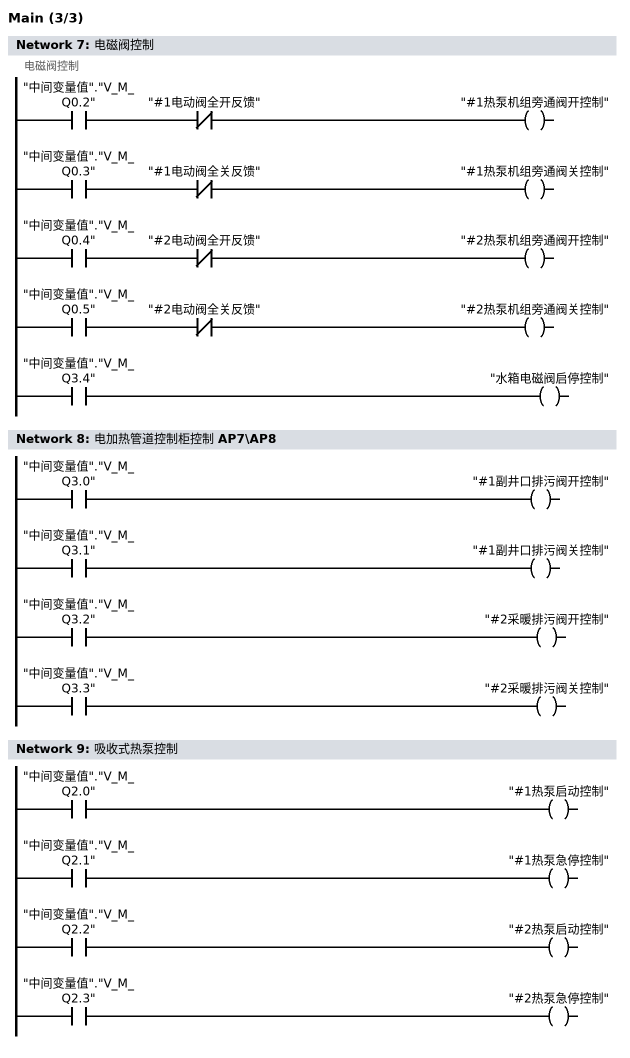
   RUNG wire#powerrail
      Contact( "中间变量值"."V_M_Q0.2" )
      I_Contact( "#1电动阀全开反馈" )
      Coil( "#1热泵机组旁通阀开控制" )
   END_RUNG
   RUNG wire#powerrail
      Contact( "中间变量值"."V_M_Q0.3" )
      I_Contact( "#1电动阀全关反馈" )
      Coil( "#1热泵机组旁通阀关控制" )
   END_RUNG
   RUNG wire#powerrail
      Contact( "中间变量值"."V_M_Q0.4" )
      I_Contact( "#2电动阀全开反馈" )
      Coil( "#2热泵机组旁通阀开控制" )
   END_RUNG
   RUNG wire#powerrail
      Contact( "中间变量值"."V_M_Q0.5" )
      I_Contact( "#2电动阀全关反馈" )
      Coil( "#2热泵机组旁通阀关控制" )
   END_RUNG
   RUNG wire#powerrail
      Contact( "中间变量值"."V_M_Q3.4" )
      Coil( "水箱电磁阀启停控制" )
   END_RUNG
   // the same network as SCL:
   "#1热泵机组旁通阀开控制" := "中间变量值"."V_M_Q0.2" AND NOT "#1电动阀全开反馈";
   "#1热泵机组旁通阀关控制" := "中间变量值"."V_M_Q0.3" AND NOT "#1电动阀全关反馈";
   "#2热泵机组旁通阀开控制" := "中间变量值"."V_M_Q0.4" AND NOT "#2电动阀全开反馈";
   "#2热泵机组旁通阀关控制" := "中间变量值"."V_M_Q0.5" AND NOT "#2电动阀全关反馈";
   "水箱电磁阀启停控制" := "中间变量值"."V_M_Q3.4";
END_REGION

REGION Network 8: 电加热管道控制柜控制 AP7\AP8
   RUNG wire#powerrail
      Contact( "中间变量值"."V_M_Q3.0" )
      Coil( "#1副井口排污阀开控制" )
   END_RUNG
   RUNG wire#powerrail
      Contact( "中间变量值"."V_M_Q3.1" )
      Coil( "#1副井口排污阀关控制" )
   END_RUNG
   RUNG wire#powerrail
      Contact( "中间变量值"."V_M_Q3.2" )
      Coil( "#2采暖排污阀开控制" )
   END_RUNG
   RUNG wire#powerrail
      Contact( "中间变量值"."V_M_Q3.3" )
      Coil( "#2采暖排污阀关控制" )
   END_RUNG
   // the same network as SCL:
   "#1副井口排污阀开控制" := "中间变量值"."V_M_Q3.0";
   "#1副井口排污阀关控制" := "中间变量值"."V_M_Q3.1";
   "#2采暖排污阀开控制" := "中间变量值"."V_M_Q3.2";
   "#2采暖排污阀关控制" := "中间变量值"."V_M_Q3.3";
END_REGION

REGION Network 9: 吸收式热泵控制
   RUNG wire#powerrail
      Contact( "中间变量值"."V_M_Q2.0" )
      Coil( "#1热泵启动控制" )
   END_RUNG
   RUNG wire#powerrail
      Contact( "中间变量值"."V_M_Q2.1" )
      Coil( "#1热泵急停控制" )
   END_RUNG
   RUNG wire#powerrail
      Contact( "中间变量值"."V_M_Q2.2" )
      Coil( "#2热泵启动控制" )
   END_RUNG
   RUNG wire#powerrail
      Contact( "中间变量值"."V_M_Q2.3" )
      Coil( "#2热泵急停控制" )
   END_RUNG
   // the same network as SCL:
   "#1热泵启动控制" := "中间变量值"."V_M_Q2.0";
   "#1热泵急停控制" := "中间变量值"."V_M_Q2.1";
   "#2热泵启动控制" := "中间变量值"."V_M_Q2.2";
   "#2热泵急停控制" := "中间变量值"."V_M_Q2.3";
END_REGION
END_ORGANIZATION_BLOCK

ORGANIZATION_BLOCK "OnTimer_模拟量定时采集"   // OB30, LAD, CyclicInterrupt
{ S7_Optimized_Access := 'TRUE' }
VERSION : 0.1
   VAR_INPUT
      Initial_Call : Bool;   // Initial call of this OB
      Event_Count : Int;   // Events discarded
   END_VAR
   VAR_TEMP   // added for the SCL form of the ladder/FBD networks
      _w1 : Bool;
      _w2 : Bool;
      _w3 : Bool;
      _w4 : Bool;
      _w5 : Bool;
      _w6 : Bool;
      _w7 : Bool;
      _w8 : Bool;
   END_VAR
BEGIN

REGION Network 2
   // 压力值获取
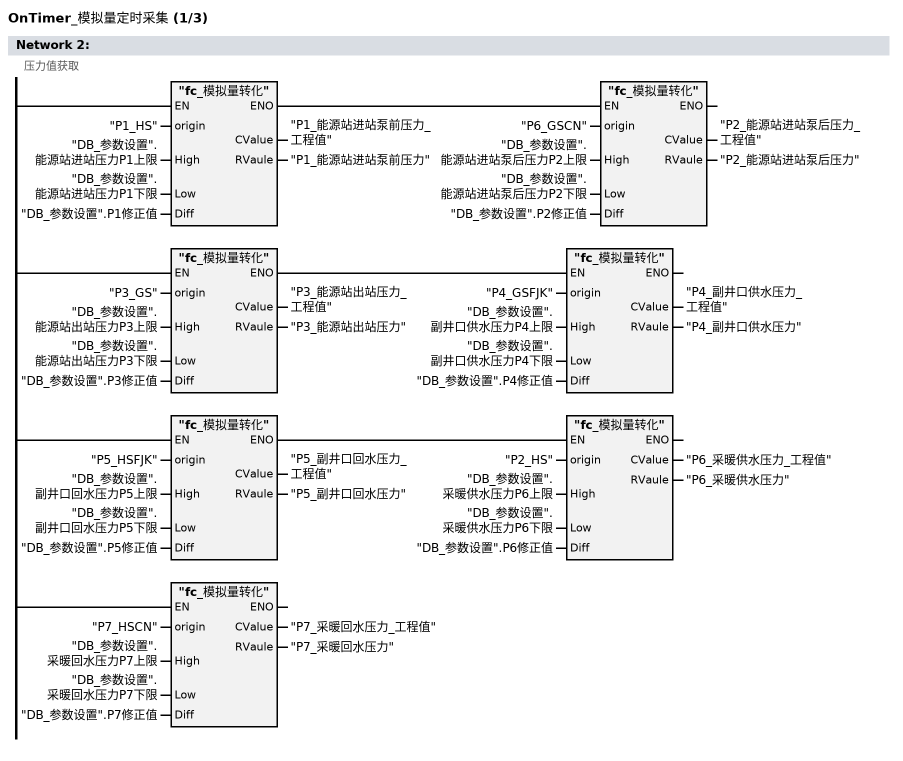
   RUNG wire#powerrail
      "fc_模拟量转化"(origin := "P1_HS", High := "DB_参数设置".能源站进站压力P1上限, Low := "DB_参数设置".能源站进站压力P1下限, Diff := "DB_参数设置".P1修正值, CValue => "P1_能源站进站泵前压力_工程值", RVaule => "P1_能源站进站泵前压力")
      "fc_模拟量转化"(origin := "P6_GSCN", High := "DB_参数设置".能源站进站泵后压力P2上限, Low := "DB_参数设置".能源站进站泵后压力P2下限, Diff := "DB_参数设置".P2修正值, CValue => "P2_能源站进站泵后压力_工程值", RVaule => "P2_能源站进站泵后压力")
   END_RUNG
   RUNG wire#powerrail
      "fc_模拟量转化"(origin := "P3_GS", High := "DB_参数设置".能源站出站压力P3上限, Low := "DB_参数设置".能源站出站压力P3下限, Diff := "DB_参数设置".P3修正值, CValue => "P3_能源站出站压力_工程值", RVaule => "P3_能源站出站压力")
      "fc_模拟量转化"(origin := "P4_GSFJK", High := "DB_参数设置".副井口供水压力P4上限, Low := "DB_参数设置".副井口供水压力P4下限, Diff := "DB_参数设置".P4修正值, CValue => "P4_副井口供水压力_工程值", RVaule => "P4_副井口供水压力")
   END_RUNG
   RUNG wire#powerrail
      "fc_模拟量转化"(origin := "P5_HSFJK", High := "DB_参数设置".副井口回水压力P5上限, Low := "DB_参数设置".副井口回水压力P5下限, Diff := "DB_参数设置".P5修正值, CValue => "P5_副井口回水压力_工程值", RVaule => "P5_副井口回水压力")
      "fc_模拟量转化"(origin := "P2_HS", High := "DB_参数设置".采暖供水压力P6上限, Low := "DB_参数设置".采暖供水压力P6下限, Diff := "DB_参数设置".P6修正值, CValue => "P6_采暖供水压力_工程值", RVaule => "P6_采暖供水压力")
   END_RUNG
   RUNG wire#powerrail
      "fc_模拟量转化"(origin := "P7_HSCN", High := "DB_参数设置".采暖回水压力P7上限, Low := "DB_参数设置".采暖回水压力P7下限, Diff := "DB_参数设置".P7修正值, CValue => "P7_采暖回水压力_工程值", RVaule => "P7_采暖回水压力")
   END_RUNG
   // the same network as SCL:
   "fc_模拟量转化"(origin := "P1_HS",
              High := "DB_参数设置".能源站进站压力P1上限,
              Low := "DB_参数设置".能源站进站压力P1下限,
              Diff := "DB_参数设置".P1修正值,
              CValue => "P1_能源站进站泵前压力_工程值",
              RVaule => "P1_能源站进站泵前压力",
              ENO => #_w1);
   IF #_w1 THEN
       "fc_模拟量转化"(origin := "P6_GSCN",
                  High := "DB_参数设置".能源站进站泵后压力P2上限,
                  Low := "DB_参数设置".能源站进站泵后压力P2下限,
                  Diff := "DB_参数设置".P2修正值,
                  CValue => "P2_能源站进站泵后压力_工程值",
                  RVaule => "P2_能源站进站泵后压力");
   END_IF;
   "fc_模拟量转化"(origin := "P3_GS",
              High := "DB_参数设置".能源站出站压力P3上限,
              Low := "DB_参数设置".能源站出站压力P3下限,
              Diff := "DB_参数设置".P3修正值,
              CValue => "P3_能源站出站压力_工程值",
              RVaule => "P3_能源站出站压力",
              ENO => #_w2);
   IF #_w2 THEN
       "fc_模拟量转化"(origin := "P4_GSFJK",
                  High := "DB_参数设置".副井口供水压力P4上限,
                  Low := "DB_参数设置".副井口供水压力P4下限,
                  Diff := "DB_参数设置".P4修正值,
                  CValue => "P4_副井口供水压力_工程值",
                  RVaule => "P4_副井口供水压力");
   END_IF;
   "fc_模拟量转化"(origin := "P5_HSFJK",
              High := "DB_参数设置".副井口回水压力P5上限,
              Low := "DB_参数设置".副井口回水压力P5下限,
              Diff := "DB_参数设置".P5修正值,
              CValue => "P5_副井口回水压力_工程值",
              RVaule => "P5_副井口回水压力",
              ENO => #_w3);
   IF #_w3 THEN
       "fc_模拟量转化"(origin := "P2_HS",
                  High := "DB_参数设置".采暖供水压力P6上限,
                  Low := "DB_参数设置".采暖供水压力P6下限,
                  Diff := "DB_参数设置".P6修正值,
                  CValue => "P6_采暖供水压力_工程值",
                  RVaule => "P6_采暖供水压力");
   END_IF;
   "fc_模拟量转化"(origin := "P7_HSCN",
              High := "DB_参数设置".采暖回水压力P7上限,
              Low := "DB_参数设置".采暖回水压力P7下限,
              Diff := "DB_参数设置".P7修正值,
              CValue => "P7_采暖回水压力_工程值",
              RVaule => "P7_采暖回水压力");
END_REGION

REGION Network 3
   // 温度T1-T12
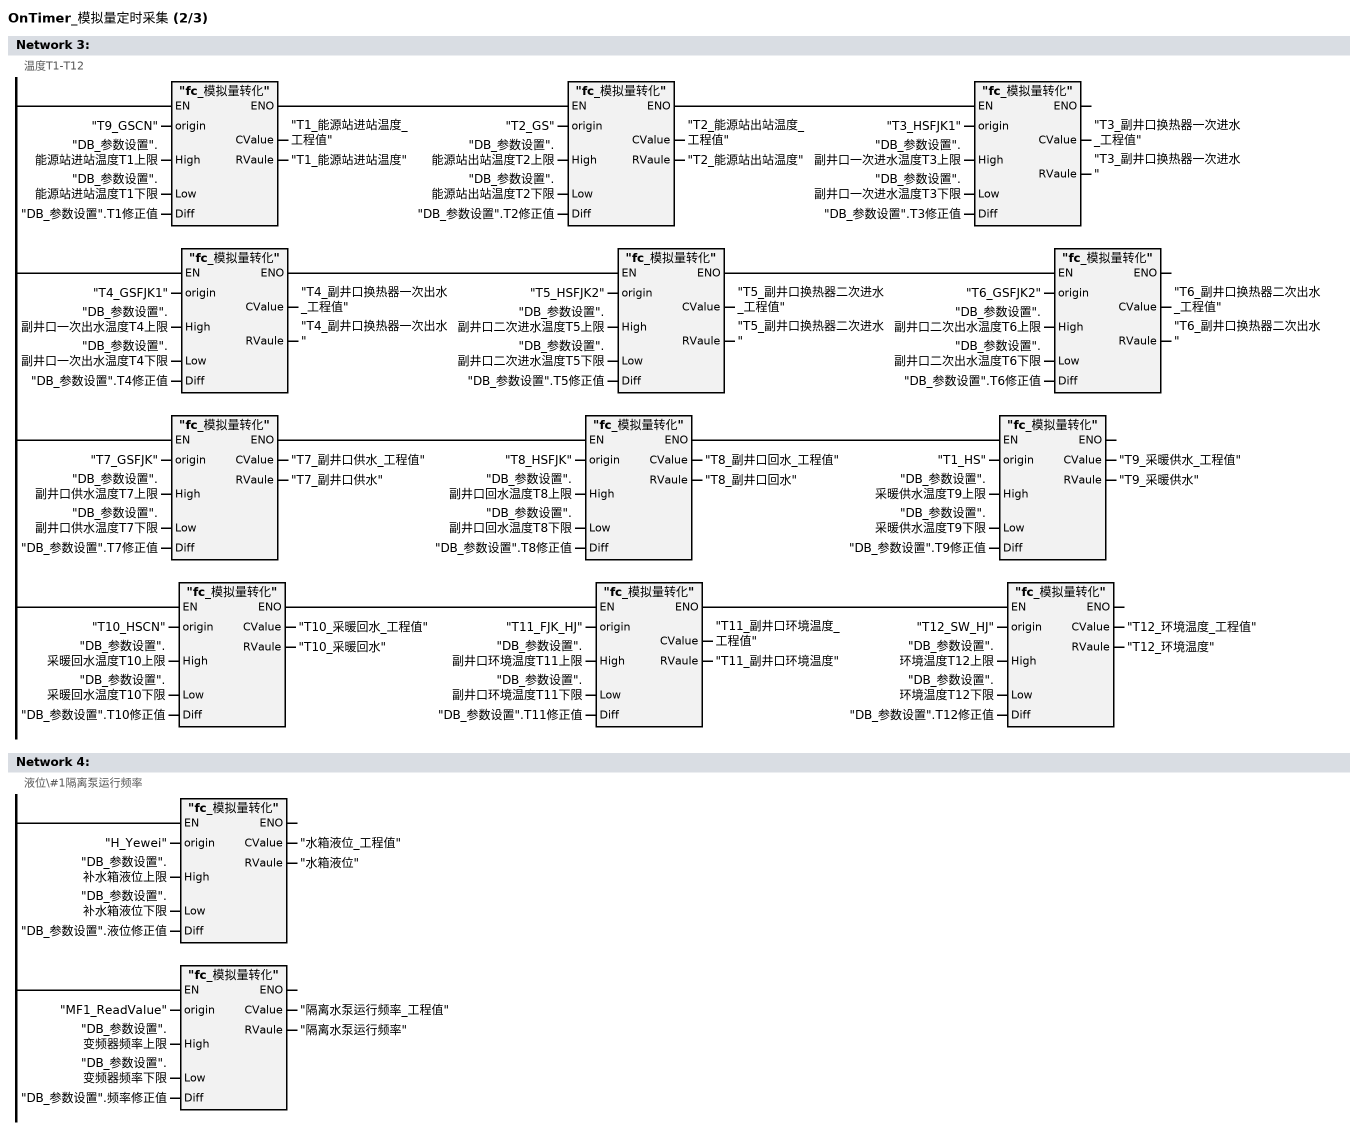
   RUNG wire#powerrail
      "fc_模拟量转化"(origin := "T9_GSCN", High := "DB_参数设置".能源站进站温度T1上限, Low := "DB_参数设置".能源站进站温度T1下限, Diff := "DB_参数设置".T1修正值, CValue => "T1_能源站进站温度_工程值", RVaule => "T1_能源站进站温度")
      "fc_模拟量转化"(origin := "T2_GS", High := "DB_参数设置".能源站出站温度T2上限, Low := "DB_参数设置".能源站出站温度T2下限, Diff := "DB_参数设置".T2修正值, CValue => "T2_能源站出站温度_工程值", RVaule => "T2_能源站出站温度")
      "fc_模拟量转化"(origin := "T3_HSFJK1", High := "DB_参数设置".副井口一次进水温度T3上限, Low := "DB_参数设置".副井口一次进水温度T3下限, Diff := "DB_参数设置".T3修正值, CValue => "T3_副井口换热器一次进水_工程值", RVaule => "T3_副井口换热器一次进水")
   END_RUNG
   RUNG wire#powerrail
      "fc_模拟量转化"(origin := "T4_GSFJK1", High := "DB_参数设置".副井口一次出水温度T4上限, Low := "DB_参数设置".副井口一次出水温度T4下限, Diff := "DB_参数设置".T4修正值, CValue => "T4_副井口换热器一次出水_工程值", RVaule => "T4_副井口换热器一次出水")
      "fc_模拟量转化"(origin := "T5_HSFJK2", High := "DB_参数设置".副井口二次进水温度T5上限, Low := "DB_参数设置".副井口二次进水温度T5下限, Diff := "DB_参数设置".T5修正值, CValue => "T5_副井口换热器二次进水_工程值", RVaule => "T5_副井口换热器二次进水")
      "fc_模拟量转化"(origin := "T6_GSFJK2", High := "DB_参数设置".副井口二次出水温度T6上限, Low := "DB_参数设置".副井口二次出水温度T6下限, Diff := "DB_参数设置".T6修正值, CValue => "T6_副井口换热器二次出水_工程值", RVaule => "T6_副井口换热器二次出水")
   END_RUNG
   RUNG wire#powerrail
      "fc_模拟量转化"(origin := "T7_GSFJK", High := "DB_参数设置".副井口供水温度T7上限, Low := "DB_参数设置".副井口供水温度T7下限, Diff := "DB_参数设置".T7修正值, CValue => "T7_副井口供水_工程值", RVaule => "T7_副井口供水")
      "fc_模拟量转化"(origin := "T8_HSFJK", High := "DB_参数设置".副井口回水温度T8上限, Low := "DB_参数设置".副井口回水温度T8下限, Diff := "DB_参数设置".T8修正值, CValue => "T8_副井口回水_工程值", RVaule => "T8_副井口回水")
      "fc_模拟量转化"(origin := "T1_HS", High := "DB_参数设置".采暖供水温度T9上限, Low := "DB_参数设置".采暖供水温度T9下限, Diff := "DB_参数设置".T9修正值, CValue => "T9_采暖供水_工程值", RVaule => "T9_采暖供水")
   END_RUNG
   RUNG wire#powerrail
      "fc_模拟量转化"(origin := "T10_HSCN", High := "DB_参数设置".采暖回水温度T10上限, Low := "DB_参数设置".采暖回水温度T10下限, Diff := "DB_参数设置".T10修正值, CValue => "T10_采暖回水_工程值", RVaule => "T10_采暖回水")
      "fc_模拟量转化"(origin := "T11_FJK_HJ", High := "DB_参数设置".副井口环境温度T11上限, Low := "DB_参数设置".副井口环境温度T11下限, Diff := "DB_参数设置".T11修正值, CValue => "T11_副井口环境温度_工程值", RVaule => "T11_副井口环境温度")
      "fc_模拟量转化"(origin := "T12_SW_HJ", High := "DB_参数设置".环境温度T12上限, Low := "DB_参数设置".环境温度T12下限, Diff := "DB_参数设置".T12修正值, CValue => "T12_环境温度_工程值", RVaule => "T12_环境温度")
   END_RUNG
   // the same network as SCL:
   "fc_模拟量转化"(origin := "T9_GSCN",
              High := "DB_参数设置".能源站进站温度T1上限,
              Low := "DB_参数设置".能源站进站温度T1下限,
              Diff := "DB_参数设置".T1修正值,
              CValue => "T1_能源站进站温度_工程值",
              RVaule => "T1_能源站进站温度",
              ENO => #_w1);
   "fc_模拟量转化"(EN := #_w1,
              origin := "T2_GS",
              High := "DB_参数设置".能源站出站温度T2上限,
              Low := "DB_参数设置".能源站出站温度T2下限,
              Diff := "DB_参数设置".T2修正值,
              CValue => "T2_能源站出站温度_工程值",
              RVaule => "T2_能源站出站温度",
              ENO => #_w2);
   IF #_w2 THEN
       "fc_模拟量转化"(origin := "T3_HSFJK1",
                  High := "DB_参数设置".副井口一次进水温度T3上限,
                  Low := "DB_参数设置".副井口一次进水温度T3下限,
                  Diff := "DB_参数设置".T3修正值,
                  CValue => "T3_副井口换热器一次进水_工程值",
                  RVaule => "T3_副井口换热器一次进水");
   END_IF;
   "fc_模拟量转化"(origin := "T4_GSFJK1",
              High := "DB_参数设置".副井口一次出水温度T4上限,
              Low := "DB_参数设置".副井口一次出水温度T4下限,
              Diff := "DB_参数设置".T4修正值,
              CValue => "T4_副井口换热器一次出水_工程值",
              RVaule => "T4_副井口换热器一次出水",
              ENO => #_w3);
   "fc_模拟量转化"(EN := #_w3,
              origin := "T5_HSFJK2",
              High := "DB_参数设置".副井口二次进水温度T5上限,
              Low := "DB_参数设置".副井口二次进水温度T5下限,
              Diff := "DB_参数设置".T5修正值,
              CValue => "T5_副井口换热器二次进水_工程值",
              RVaule => "T5_副井口换热器二次进水",
              ENO => #_w4);
   IF #_w4 THEN
       "fc_模拟量转化"(origin := "T6_GSFJK2",
                  High := "DB_参数设置".副井口二次出水温度T6上限,
                  Low := "DB_参数设置".副井口二次出水温度T6下限,
                  Diff := "DB_参数设置".T6修正值,
                  CValue => "T6_副井口换热器二次出水_工程值",
                  RVaule => "T6_副井口换热器二次出水");
   END_IF;
   "fc_模拟量转化"(origin := "T7_GSFJK",
              High := "DB_参数设置".副井口供水温度T7上限,
              Low := "DB_参数设置".副井口供水温度T7下限,
              Diff := "DB_参数设置".T7修正值,
              CValue => "T7_副井口供水_工程值",
              RVaule => "T7_副井口供水",
              ENO => #_w5);
   "fc_模拟量转化"(EN := #_w5,
              origin := "T8_HSFJK",
              High := "DB_参数设置".副井口回水温度T8上限,
              Low := "DB_参数设置".副井口回水温度T8下限,
              Diff := "DB_参数设置".T8修正值,
              CValue => "T8_副井口回水_工程值",
              RVaule => "T8_副井口回水",
              ENO => #_w6);
   IF #_w6 THEN
       "fc_模拟量转化"(origin := "T1_HS",
                  High := "DB_参数设置".采暖供水温度T9上限,
                  Low := "DB_参数设置".采暖供水温度T9下限,
                  Diff := "DB_参数设置".T9修正值,
                  CValue => "T9_采暖供水_工程值",
                  RVaule => "T9_采暖供水");
   END_IF;
   "fc_模拟量转化"(origin := "T10_HSCN",
              High := "DB_参数设置".采暖回水温度T10上限,
              Low := "DB_参数设置".采暖回水温度T10下限,
              Diff := "DB_参数设置".T10修正值,
              CValue => "T10_采暖回水_工程值",
              RVaule => "T10_采暖回水",
              ENO => #_w7);
   "fc_模拟量转化"(EN := #_w7,
              origin := "T11_FJK_HJ",
              High := "DB_参数设置".副井口环境温度T11上限,
              Low := "DB_参数设置".副井口环境温度T11下限,
              Diff := "DB_参数设置".T11修正值,
              CValue => "T11_副井口环境温度_工程值",
              RVaule => "T11_副井口环境温度",
              ENO => #_w8);
   IF #_w8 THEN
       "fc_模拟量转化"(origin := "T12_SW_HJ",
                  High := "DB_参数设置".环境温度T12上限,
                  Low := "DB_参数设置".环境温度T12下限,
                  Diff := "DB_参数设置".T12修正值,
                  CValue => "T12_环境温度_工程值",
                  RVaule => "T12_环境温度");
   END_IF;
END_REGION

REGION Network 4
   // 液位\#1隔离泵运行频率
   RUNG wire#powerrail
      "fc_模拟量转化"(origin := "H_Yewei", High := "DB_参数设置".补水箱液位上限, Low := "DB_参数设置".补水箱液位下限, Diff := "DB_参数设置".液位修正值, CValue => "水箱液位_工程值", RVaule => "水箱液位")
   END_RUNG
   RUNG wire#powerrail
      "fc_模拟量转化"(origin := "MF1_ReadValue", High := "DB_参数设置".变频器频率上限, Low := "DB_参数设置".变频器频率下限, Diff := "DB_参数设置".频率修正值, CValue => "隔离水泵运行频率_工程值", RVaule => "隔离水泵运行频率")
   END_RUNG
   // the same network as SCL:
   "fc_模拟量转化"(origin := "H_Yewei",
              High := "DB_参数设置".补水箱液位上限,
              Low := "DB_参数设置".补水箱液位下限,
              Diff := "DB_参数设置".液位修正值,
              CValue => "水箱液位_工程值",
              RVaule => "水箱液位");
   "fc_模拟量转化"(origin := "MF1_ReadValue",
              High := "DB_参数设置".变频器频率上限,
              Low := "DB_参数设置".变频器频率下限,
              Diff := "DB_参数设置".频率修正值,
              CValue => "隔离水泵运行频率_工程值",
              RVaule => "隔离水泵运行频率");
END_REGION

REGION Network 5
   // 变频器设置频率
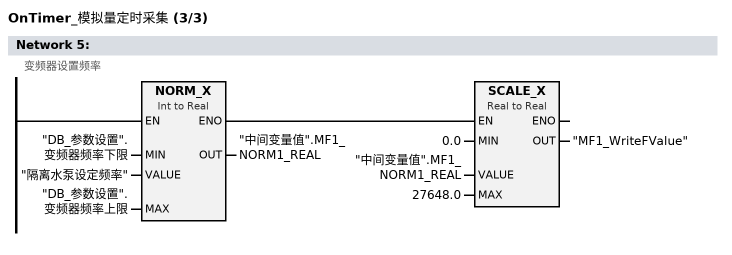
   RUNG wire#powerrail
      { S7_Templates := "[SrcType := Int, DestType := Real]" } Normalize(min := "DB_参数设置".变频器频率下限, value := "隔离水泵设定频率", max := "DB_参数设置".变频器频率上限, out => "中间变量值".MF1_NORM1_REAL)
      { S7_Templates := "[SrcType := Real, DestType := Real]" } Scale(min := 0.0, value := "中间变量值".MF1_NORM1_REAL, max := 27648.0, out => "MF1_WriteFValue")
   END_RUNG
   // the same network as SCL:
   "中间变量值".MF1_NORM1_REAL := NORM_X(MIN := "DB_参数设置".变频器频率下限, VALUE := "隔离水泵设定频率", MAX := "DB_参数设置".变频器频率上限);
   "MF1_WriteFValue" := SCALE_X(MIN := 0.0, VALUE := "中间变量值".MF1_NORM1_REAL, MAX := 27648.0);
END_REGION
END_ORGANIZATION_BLOCK

ORGANIZATION_BLOCK "Interrupt_1Min"   // OB31, LAD, CyclicInterrupt
{ S7_Optimized_Access := 'TRUE' }
VERSION : 0.1
   VAR_INPUT
      Initial_Call : Bool;   // Initial call of this OB
      Event_Count : Int;   // Events discarded
   END_VAR
BEGIN

REGION Network 1
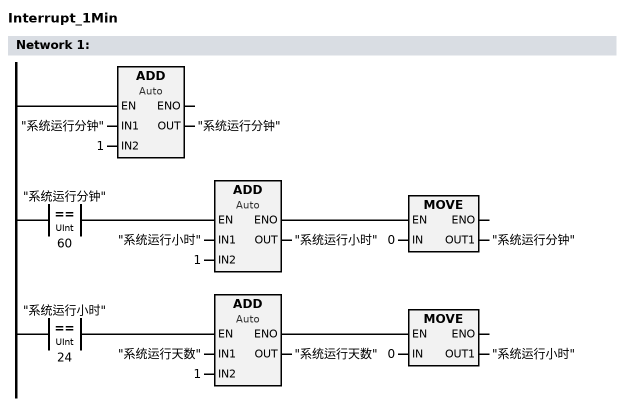
   RUNG wire#powerrail
      Add(in1 := "系统运行分钟", in2 := 1, out => "系统运行分钟")
   END_RUNG
   RUNG wire#powerrail
      { S7_Templates := "SrcType := UInt" } EQ_Contact(in1 := "系统运行分钟", in2 := 60)
      Add(in1 := "系统运行小时", in2 := 1, out => "系统运行小时")
      Move(in := 0, out1 => "系统运行分钟")
   END_RUNG
   RUNG wire#powerrail
      { S7_Templates := "SrcType := UInt" } EQ_Contact(in1 := "系统运行小时", in2 := 24)
      Add(in1 := "系统运行天数", in2 := 1, out => "系统运行天数")
      Move(in := 0, out1 => "系统运行小时")
   END_RUNG
   // the same network as SCL:
   "系统运行分钟" := "系统运行分钟" + 1;
   IF "系统运行分钟" = 60 THEN
       "系统运行小时" := "系统运行小时" + 1;
       "系统运行分钟" := 0;
   END_IF;
   IF "系统运行小时" = 24 THEN
       "系统运行天数" := "系统运行天数" + 1;
       "系统运行小时" := 0;
   END_IF;
END_REGION
END_ORGANIZATION_BLOCK

ORGANIZATION_BLOCK "Pull or plug of modules"   // OB83, LAD, PullPlug
{ S7_Optimized_Access := 'TRUE' }
VERSION : 0.1
   VAR_INPUT
      LADDR : Hw_Io;   // Hardware identifier
      Event_Class : Byte;   // 16#38/39: module inserted, removed
      Fault_ID : Byte;   // Fault identifier
   END_VAR
BEGIN
END_ORGANIZATION_BLOCK

ORGANIZATION_BLOCK "Rack or station failure"   // OB86, LAD, RackStationFailure
{ S7_Optimized_Access := 'TRUE' }
VERSION : 0.1
   VAR_INPUT
      LADDR : Hw_Device;   // Hardware identifier
      Event_Class : Byte;   // Event class
      Fault_ID : Byte;   // Fault identifier
   END_VAR
BEGIN
END_ORGANIZATION_BLOCK

ORGANIZATION_BLOCK "Startup"   // OB100, LAD, Startup
TITLE = "Complete Restart"
{ S7_Optimized_Access := 'TRUE' }
VERSION : 0.1
   VAR_INPUT
      LostRetentive : Bool;   // True if retentive data are lost
      LostRTC : Bool;   // True if date and time are lost
   END_VAR
BEGIN
END_ORGANIZATION_BLOCK

ORGANIZATION_BLOCK "sub_报警处理"   // OB123, LAD, ProgramCycle
TITLE = "Main Program Sweep (Cycle)"
{ S7_Optimized_Access := 'TRUE' }
VERSION : 0.1
   VAR_INPUT
      Initial_Call : Bool;   // Initial call of this OB
      Remanence : Bool;   // =True, if remanent data are available
   END_VAR
   VAR_TEMP   // added for the SCL form of the ladder/FBD networks
      _w1 : Bool;
      _w2 : Bool;
      _w3 : Bool;
      _w4 : Bool;
   END_VAR
BEGIN

REGION Network 1: 压力异常报警1
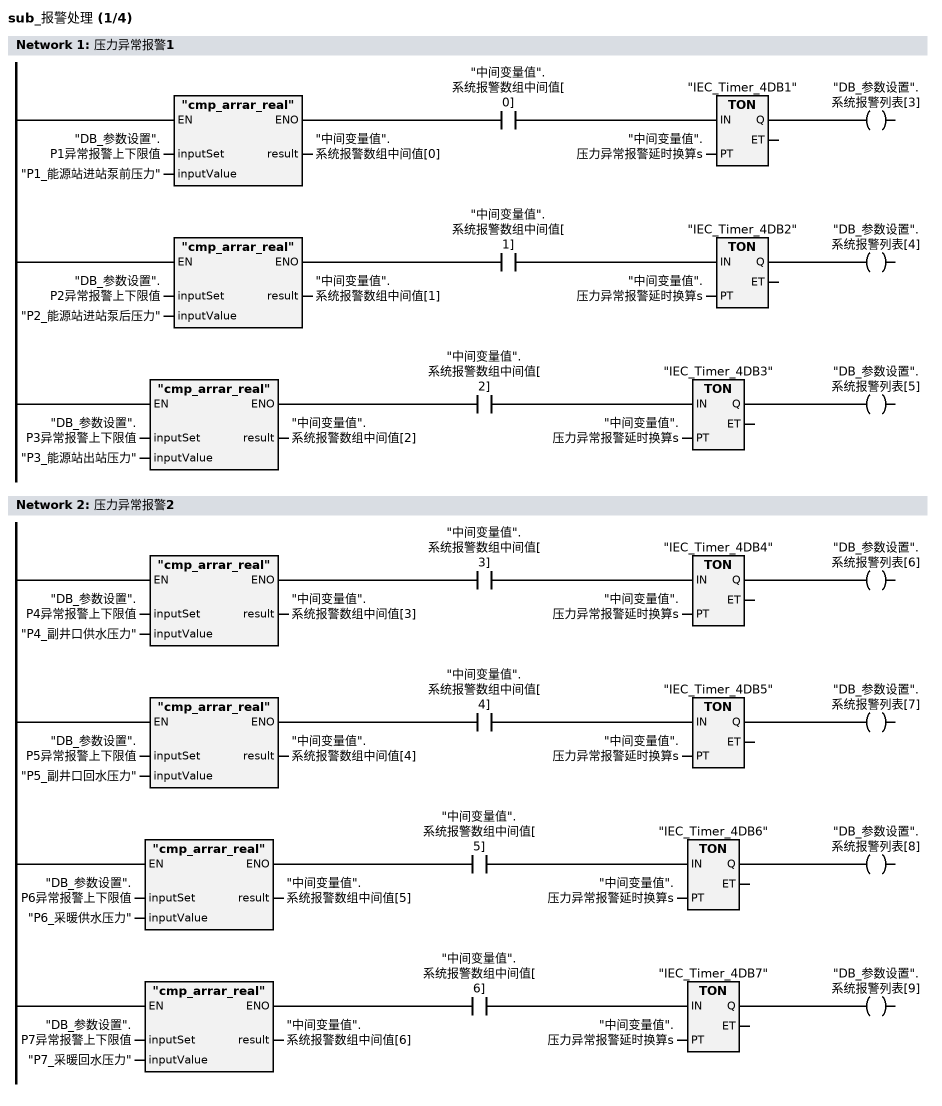
   "cmp_arrar_real"(inputSet := "DB_参数设置".P1异常报警上下限值,
                    inputValue := "P1_能源站进站泵前压力",
                    result => "中间变量值".系统报警数组中间值[0],
                    ENO => #_w1);
   "IEC_Timer_4DB1".TON(IN := #_w1 AND "中间变量值".系统报警数组中间值[0], PT := "中间变量值".压力异常报警延时换算s);
   "DB_参数设置".系统报警列表[3] := "IEC_Timer_4DB1".Q;
   "cmp_arrar_real"(inputSet := "DB_参数设置".P2异常报警上下限值,
                    inputValue := "P2_能源站进站泵后压力",
                    result => "中间变量值".系统报警数组中间值[1],
                    ENO => #_w2);
   "IEC_Timer_4DB2".TON(IN := #_w2 AND "中间变量值".系统报警数组中间值[1], PT := "中间变量值".压力异常报警延时换算s);
   "DB_参数设置".系统报警列表[4] := "IEC_Timer_4DB2".Q;
   "cmp_arrar_real"(inputSet := "DB_参数设置".P3异常报警上下限值,
                    inputValue := "P3_能源站出站压力",
                    result => "中间变量值".系统报警数组中间值[2],
                    ENO => #_w3);
   "IEC_Timer_4DB3".TON(IN := #_w3 AND "中间变量值".系统报警数组中间值[2], PT := "中间变量值".压力异常报警延时换算s);
   "DB_参数设置".系统报警列表[5] := "IEC_Timer_4DB3".Q;
END_REGION

REGION Network 2: 压力异常报警2
   "cmp_arrar_real"(inputSet := "DB_参数设置".P4异常报警上下限值,
                    inputValue := "P4_副井口供水压力",
                    result => "中间变量值".系统报警数组中间值[3],
                    ENO => #_w1);
   "IEC_Timer_4DB4".TON(IN := #_w1 AND "中间变量值".系统报警数组中间值[3], PT := "中间变量值".压力异常报警延时换算s);
   "DB_参数设置".系统报警列表[6] := "IEC_Timer_4DB4".Q;
   "cmp_arrar_real"(inputSet := "DB_参数设置".P5异常报警上下限值,
                    inputValue := "P5_副井口回水压力",
                    result => "中间变量值".系统报警数组中间值[4],
                    ENO => #_w2);
   "IEC_Timer_4DB5".TON(IN := #_w2 AND "中间变量值".系统报警数组中间值[4], PT := "中间变量值".压力异常报警延时换算s);
   "DB_参数设置".系统报警列表[7] := "IEC_Timer_4DB5".Q;
   "cmp_arrar_real"(inputSet := "DB_参数设置".P6异常报警上下限值,
                    inputValue := "P6_采暖供水压力",
                    result => "中间变量值".系统报警数组中间值[5],
                    ENO => #_w3);
   "IEC_Timer_4DB6".TON(IN := #_w3 AND "中间变量值".系统报警数组中间值[5], PT := "中间变量值".压力异常报警延时换算s);
   "DB_参数设置".系统报警列表[8] := "IEC_Timer_4DB6".Q;
   "cmp_arrar_real"(inputSet := "DB_参数设置".P7异常报警上下限值,
                    inputValue := "P7_采暖回水压力",
                    result => "中间变量值".系统报警数组中间值[6],
                    ENO => #_w4);
   "IEC_Timer_4DB7".TON(IN := #_w4 AND "中间变量值".系统报警数组中间值[6], PT := "中间变量值".压力异常报警延时换算s);
   "DB_参数设置".系统报警列表[9] := "IEC_Timer_4DB7".Q;
END_REGION

REGION Network 3: 温度 异常报警
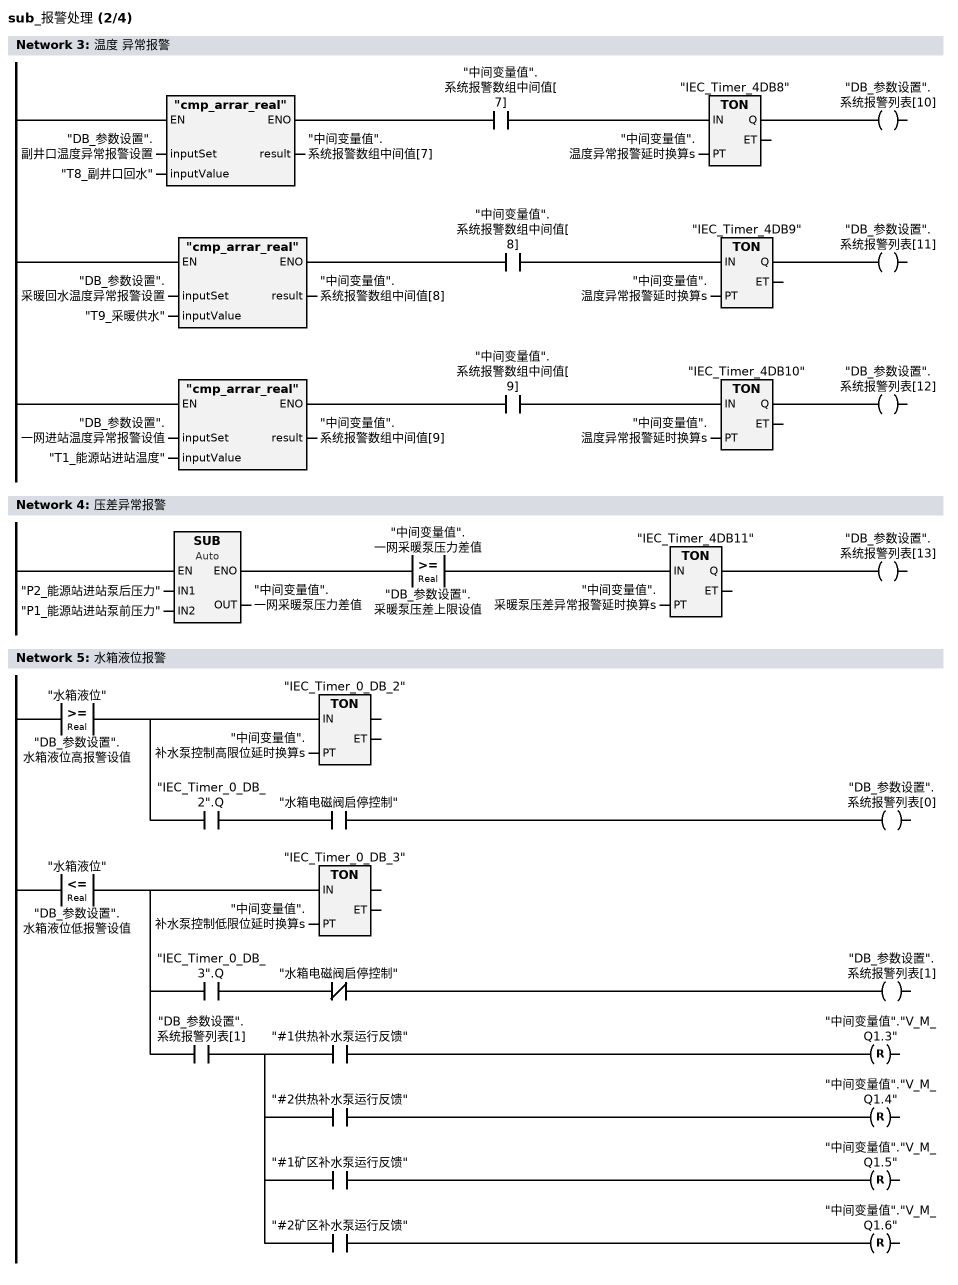
   "cmp_arrar_real"(inputSet := "DB_参数设置".副井口温度异常报警设置,
                    inputValue := "T8_副井口回水",
                    result => "中间变量值".系统报警数组中间值[7],
                    ENO => #_w1);
   "IEC_Timer_4DB8".TON(IN := #_w1 AND "中间变量值".系统报警数组中间值[7], PT := "中间变量值".温度异常报警延时换算s);
   "DB_参数设置".系统报警列表[10] := "IEC_Timer_4DB8".Q;
   "cmp_arrar_real"(inputSet := "DB_参数设置".采暖回水温度异常报警设置,
                    inputValue := "T9_采暖供水",
                    result => "中间变量值".系统报警数组中间值[8],
                    ENO => #_w2);
   "IEC_Timer_4DB9".TON(IN := #_w2 AND "中间变量值".系统报警数组中间值[8], PT := "中间变量值".温度异常报警延时换算s);
   "DB_参数设置".系统报警列表[11] := "IEC_Timer_4DB9".Q;
   "cmp_arrar_real"(inputSet := "DB_参数设置".一网进站温度异常报警设值,
                    inputValue := "T1_能源站进站温度",
                    result => "中间变量值".系统报警数组中间值[9],
                    ENO => #_w3);
   "IEC_Timer_4DB10".TON(IN := #_w3 AND "中间变量值".系统报警数组中间值[9], PT := "中间变量值".温度异常报警延时换算s);
   "DB_参数设置".系统报警列表[12] := "IEC_Timer_4DB10".Q;
END_REGION

REGION Network 4: 压差异常报警
   "中间变量值".一网采暖泵压力差值 := "P2_能源站进站泵后压力" - "P1_能源站进站泵前压力";
   "IEC_Timer_4DB11".TON(IN := "中间变量值".一网采暖泵压力差值 >= "DB_参数设置".采暖泵压差上限设值, PT := "中间变量值".采暖泵压差异常报警延时换算s);
   "DB_参数设置".系统报警列表[13] := "IEC_Timer_4DB11".Q;
END_REGION

REGION Network 5: 水箱液位报警
   #_w1 := "水箱液位" >= "DB_参数设置".水箱液位高报警设值;
   "IEC_Timer_0_DB_2".TON(IN := #_w1, PT := "中间变量值".补水泵控制高限位延时换算s);
   "DB_参数设置".系统报警列表[0] := #_w1 AND "IEC_Timer_0_DB_2".Q AND "水箱电磁阀启停控制";
   #_w2 := "水箱液位" <= "DB_参数设置".水箱液位低报警设值;
   "IEC_Timer_0_DB_3".TON(IN := #_w2, PT := "中间变量值".补水泵控制低限位延时换算s);
   "DB_参数设置".系统报警列表[1] := #_w2 AND "IEC_Timer_0_DB_3".Q AND NOT "水箱电磁阀启停控制";
   #_w3 := #_w2 AND "DB_参数设置".系统报警列表[1];
   IF #_w3 AND "#1供热补水泵运行反馈" THEN "中间变量值"."V_M_Q1.3" := FALSE; END_IF;
   IF #_w3 AND "#2供热补水泵运行反馈" THEN "中间变量值"."V_M_Q1.4" := FALSE; END_IF;
   IF #_w3 AND "#1矿区补水泵运行反馈" THEN "中间变量值"."V_M_Q1.5" := FALSE; END_IF;
   IF #_w3 AND "#2矿区补水泵运行反馈" THEN "中间变量值"."V_M_Q1.6" := FALSE; END_IF;
END_REGION

REGION Network 6: 补水参数错误检测
   // 补水参数错误检测
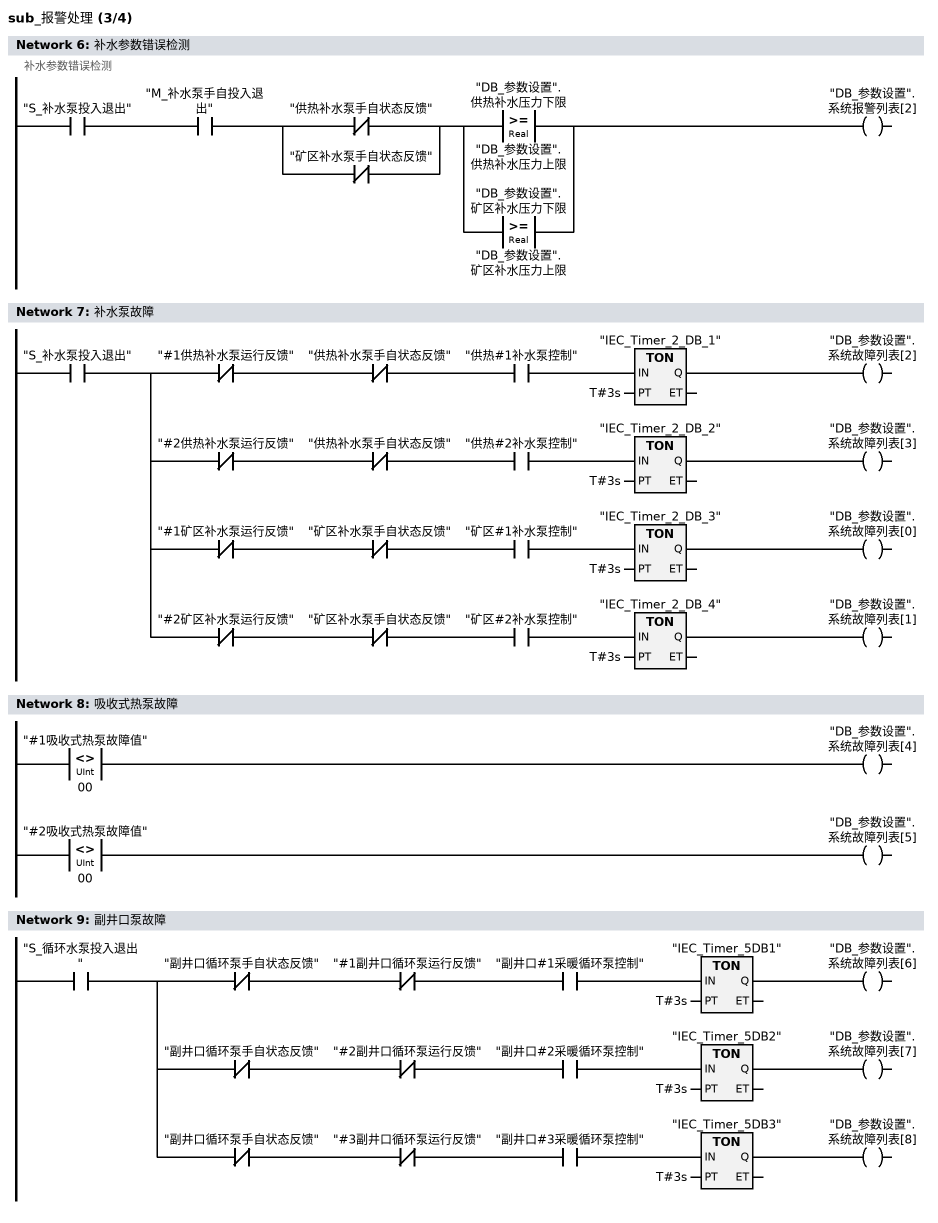
   RUNG wire#powerrail
      Contact( "S_补水泵投入退出" )
      Contact( "M_补水泵手自投入退出" )
      wire#w1
      I_Contact( "供热补水泵手自状态反馈" )
      wire#w2
      { S7_Templates := "SrcType := Real" } GE_Contact(in1 := "DB_参数设置".供热补水压力下限, in2 := "DB_参数设置".供热补水压力上限)
      wire#w3
      Coil( "DB_参数设置".系统报警列表[2] )
   END_RUNG
   RUNG wire#w1
      I_Contact( "矿区补水泵手自状态反馈" )
   END_RUNG wire#w2
   RUNG wire#w2
      { S7_Templates := "SrcType := Real" } GE_Contact(in1 := "DB_参数设置".矿区补水压力下限, in2 := "DB_参数设置".矿区补水压力上限)
   END_RUNG wire#w3
   // the same network as SCL:
   "DB_参数设置".系统报警列表[2] := "S_补水泵投入退出" AND "M_补水泵手自投入退出" AND (NOT "供热补水泵手自状态反馈" OR NOT "矿区补水泵手自状态反馈") AND (("DB_参数设置".供热补水压力下限 >= "DB_参数设置".供热补水压力上限) OR ("DB_参数设置".矿区补水压力下限 >= "DB_参数设置".矿区补水压力上限));
END_REGION

REGION Network 7: 补水泵故障
   "IEC_Timer_2_DB_1".TON(IN := "S_补水泵投入退出" AND NOT "#1供热补水泵运行反馈" AND NOT "供热补水泵手自状态反馈" AND "供热#1补水泵控制",
                          PT := T#3s);
   "DB_参数设置".系统故障列表[2] := "IEC_Timer_2_DB_1".Q;
   "IEC_Timer_2_DB_2".TON(IN := "S_补水泵投入退出" AND NOT "#2供热补水泵运行反馈" AND NOT "供热补水泵手自状态反馈" AND "供热#2补水泵控制",
                          PT := T#3s);
   "DB_参数设置".系统故障列表[3] := "IEC_Timer_2_DB_2".Q;
   "IEC_Timer_2_DB_3".TON(IN := "S_补水泵投入退出" AND NOT "#1矿区补水泵运行反馈" AND NOT "矿区补水泵手自状态反馈" AND "矿区#1补水泵控制",
                          PT := T#3s);
   "DB_参数设置".系统故障列表[0] := "IEC_Timer_2_DB_3".Q;
   "IEC_Timer_2_DB_4".TON(IN := "S_补水泵投入退出" AND NOT "#2矿区补水泵运行反馈" AND NOT "矿区补水泵手自状态反馈" AND "矿区#2补水泵控制",
                          PT := T#3s);
   "DB_参数设置".系统故障列表[1] := "IEC_Timer_2_DB_4".Q;
END_REGION

REGION Network 8: 吸收式热泵故障
   RUNG wire#powerrail
      { S7_Templates := "SrcType := UInt" } NE_Contact(in1 := "#1吸收式热泵故障值", in2 := 00)
      Coil( "DB_参数设置".系统故障列表[4] )
   END_RUNG
   RUNG wire#powerrail
      { S7_Templates := "SrcType := UInt" } NE_Contact(in1 := "#2吸收式热泵故障值", in2 := 00)
      Coil( "DB_参数设置".系统故障列表[5] )
   END_RUNG
   // the same network as SCL:
   "DB_参数设置".系统故障列表[4] := "#1吸收式热泵故障值" <> 00;
   "DB_参数设置".系统故障列表[5] := "#2吸收式热泵故障值" <> 00;
END_REGION

REGION Network 9: 副井口泵故障
   "IEC_Timer_5DB1".TON(IN := "S_循环水泵投入退出" AND NOT "副井口循环泵手自状态反馈" AND NOT "#1副井口循环泵运行反馈" AND "副井口#1采暖循环泵控制",
                        PT := T#3s);
   "DB_参数设置".系统故障列表[6] := "IEC_Timer_5DB1".Q;
   "IEC_Timer_5DB2".TON(IN := "S_循环水泵投入退出" AND NOT "副井口循环泵手自状态反馈" AND NOT "#2副井口循环泵运行反馈" AND "副井口#2采暖循环泵控制",
                        PT := T#3s);
   "DB_参数设置".系统故障列表[7] := "IEC_Timer_5DB2".Q;
   "IEC_Timer_5DB3".TON(IN := "S_循环水泵投入退出" AND NOT "副井口循环泵手自状态反馈" AND NOT "#3副井口循环泵运行反馈" AND "副井口#3采暖循环泵控制",
                        PT := T#3s);
   "DB_参数设置".系统故障列表[8] := "IEC_Timer_5DB3".Q;
END_REGION

REGION Network 10: 系统报警判断
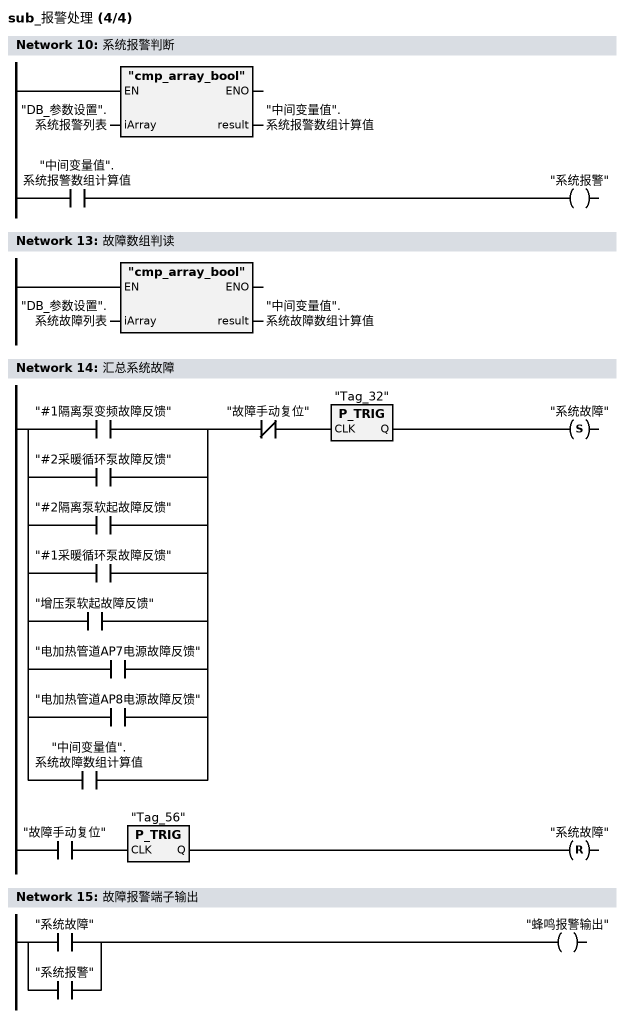
   RUNG wire#powerrail
      "cmp_array_bool"(iArray := "DB_参数设置".系统报警列表, result => "中间变量值".系统报警数组计算值)
   END_RUNG
   RUNG wire#powerrail
      Contact( "中间变量值".系统报警数组计算值 )
      Coil( "系统报警" )
   END_RUNG
   // the same network as SCL:
   "cmp_array_bool"(iArray := "DB_参数设置".系统报警列表, result => "中间变量值".系统报警数组计算值);
   "系统报警" := "中间变量值".系统报警数组计算值;
END_REGION

REGION Network 12: 系统报警
END_REGION

REGION Network 13: 故障数组判读
   RUNG wire#powerrail
      "cmp_array_bool"(iArray := "DB_参数设置".系统故障列表, result => "中间变量值".系统故障数组计算值)
   END_RUNG
   // the same network as SCL:
   "cmp_array_bool"(iArray := "DB_参数设置".系统故障列表, result => "中间变量值".系统故障数组计算值);
END_REGION

REGION Network 14: 汇总系统故障
   RUNG wire#powerrail
      Contact( "#1隔离泵变频故障反馈" )
      wire#w1
      I_Contact( "故障手动复位" )
      P_Trig( "Tag_32" )
      S_Coil( "系统故障" )
   END_RUNG
   RUNG wire#powerrail
      Contact( "#2采暖循环泵故障反馈" )
   END_RUNG wire#w1
   RUNG wire#powerrail
      Contact( "#2隔离泵软起故障反馈" )
   END_RUNG wire#w1
   RUNG wire#powerrail
      Contact( "#1采暖循环泵故障反馈" )
   END_RUNG wire#w1
   RUNG wire#powerrail
      Contact( "增压泵软起故障反馈" )
   END_RUNG wire#w1
   RUNG wire#powerrail
      Contact( "电加热管道AP7电源故障反馈" )
   END_RUNG wire#w1
   RUNG wire#powerrail
      Contact( "电加热管道AP8电源故障反馈" )
   END_RUNG wire#w1
   RUNG wire#powerrail
      Contact( "中间变量值".系统故障数组计算值 )
   END_RUNG wire#w1
   RUNG wire#powerrail
      Contact( "故障手动复位" )
      P_Trig( "Tag_56" )
      R_Coil( "系统故障" )
   END_RUNG
   // the same network as SCL:
   #_w1 := ("#1隔离泵变频故障反馈" OR "#2采暖循环泵故障反馈" OR "#2隔离泵软起故障反馈" OR "#1采暖循环泵故障反馈" OR "增压泵软起故障反馈" OR "电加热管道AP7电源故障反馈" OR "电加热管道AP8电源故障反馈" OR "中间变量值".系统故障数组计算值) AND NOT "故障手动复位";
   #_w2 := #_w1 AND NOT "Tag_32";   // rising edge
   "Tag_32" := #_w1;
   IF #_w2 THEN "系统故障" := TRUE; END_IF;
   #_w3 := "故障手动复位" AND NOT "Tag_56";   // rising edge
   "Tag_56" := "故障手动复位";
   IF #_w3 THEN "系统故障" := FALSE; END_IF;
END_REGION

REGION Network 15: 故障报警端子输出
   RUNG wire#powerrail
      Contact( "系统故障" )
      wire#w1
      Coil( "蜂鸣报警输出" )
   END_RUNG
   RUNG wire#powerrail
      Contact( "系统报警" )
   END_RUNG wire#w1
   // the same network as SCL:
   "蜂鸣报警输出" := "系统故障" OR "系统报警";
END_REGION
END_ORGANIZATION_BLOCK

ORGANIZATION_BLOCK "sub_通讯数据处理"   // OB124, LAD, ProgramCycle
TITLE = "Main Program Sweep (Cycle)"
{ S7_Optimized_Access := 'TRUE' }
VERSION : 0.1
   VAR_INPUT
      Initial_Call : Bool;   // Initial call of this OB
      Remanence : Bool;   // =True, if remanent data are available
   END_VAR
BEGIN

REGION Network 1
   // 热表瞬时流量处理
   // 单位 m3/h
END_REGION

REGION Network 2: 热表瞬时热流量处理
   // 热表瞬时热流量处理
   // 单位 kwh
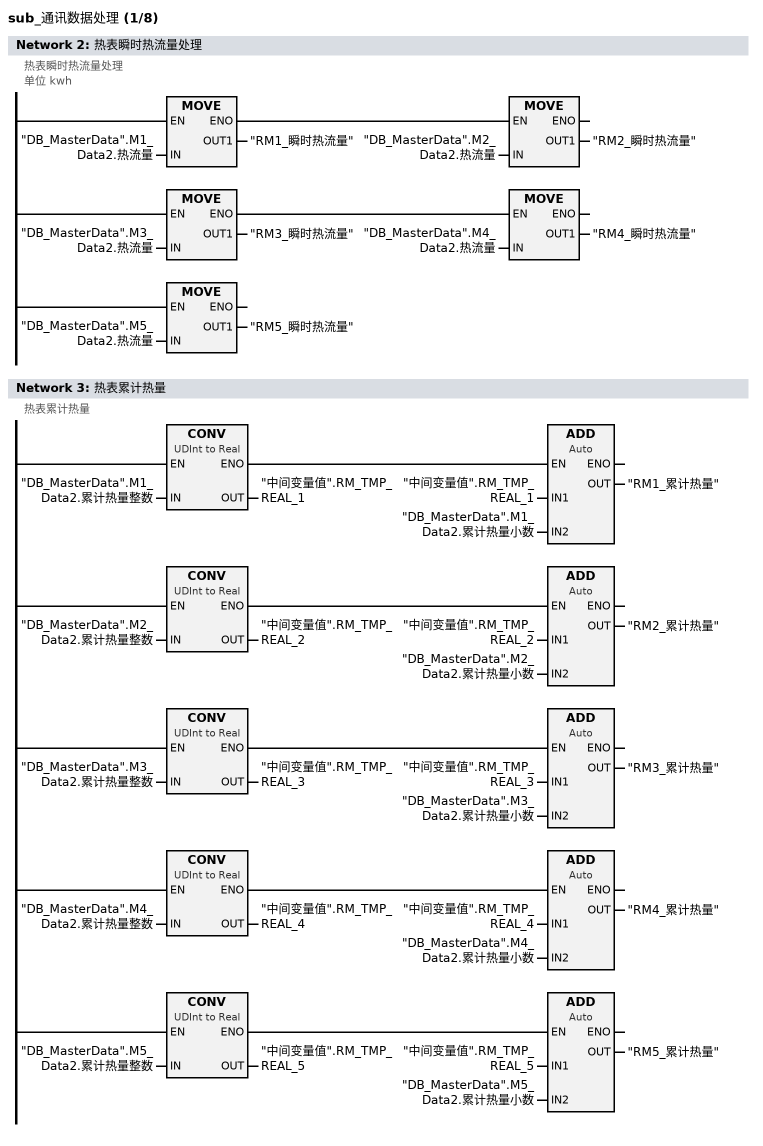
   RUNG wire#powerrail
      Move(in := "DB_MasterData".M1_Data2.热流量, out1 => "RM1_瞬时热流量")
      Move(in := "DB_MasterData".M2_Data2.热流量, out1 => "RM2_瞬时热流量")
   END_RUNG
   RUNG wire#powerrail
      Move(in := "DB_MasterData".M3_Data2.热流量, out1 => "RM3_瞬时热流量")
      Move(in := "DB_MasterData".M4_Data2.热流量, out1 => "RM4_瞬时热流量")
   END_RUNG
   RUNG wire#powerrail
      Move(in := "DB_MasterData".M5_Data2.热流量, out1 => "RM5_瞬时热流量")
   END_RUNG
   // the same network as SCL:
   "RM1_瞬时热流量" := "DB_MasterData".M1_Data2.热流量;
   "RM2_瞬时热流量" := "DB_MasterData".M2_Data2.热流量;
   "RM3_瞬时热流量" := "DB_MasterData".M3_Data2.热流量;
   "RM4_瞬时热流量" := "DB_MasterData".M4_Data2.热流量;
   "RM5_瞬时热流量" := "DB_MasterData".M5_Data2.热流量;
END_REGION

REGION Network 3: 热表累计热量
   // 热表累计热量
   RUNG wire#powerrail
      { S7_Templates := "[SrcType := UDInt, DestType := Real]" } Convert(in := "DB_MasterData".M1_Data2.累计热量整数, out => "中间变量值".RM_TMP_REAL_1)
      Add(in1 := "中间变量值".RM_TMP_REAL_1, in2 := "DB_MasterData".M1_Data2.累计热量小数, out => "RM1_累计热量")
   END_RUNG
   RUNG wire#powerrail
      { S7_Templates := "[SrcType := UDInt, DestType := Real]" } Convert(in := "DB_MasterData".M2_Data2.累计热量整数, out => "中间变量值".RM_TMP_REAL_2)
      Add(in1 := "中间变量值".RM_TMP_REAL_2, in2 := "DB_MasterData".M2_Data2.累计热量小数, out => "RM2_累计热量")
   END_RUNG
   RUNG wire#powerrail
      { S7_Templates := "[SrcType := UDInt, DestType := Real]" } Convert(in := "DB_MasterData".M3_Data2.累计热量整数, out => "中间变量值".RM_TMP_REAL_3)
      Add(in1 := "中间变量值".RM_TMP_REAL_3, in2 := "DB_MasterData".M3_Data2.累计热量小数, out => "RM3_累计热量")
   END_RUNG
   RUNG wire#powerrail
      { S7_Templates := "[SrcType := UDInt, DestType := Real]" } Convert(in := "DB_MasterData".M4_Data2.累计热量整数, out => "中间变量值".RM_TMP_REAL_4)
      Add(in1 := "中间变量值".RM_TMP_REAL_4, in2 := "DB_MasterData".M4_Data2.累计热量小数, out => "RM4_累计热量")
   END_RUNG
   RUNG wire#powerrail
      { S7_Templates := "[SrcType := UDInt, DestType := Real]" } Convert(in := "DB_MasterData".M5_Data2.累计热量整数, out => "中间变量值".RM_TMP_REAL_5)
      Add(in1 := "中间变量值".RM_TMP_REAL_5, in2 := "DB_MasterData".M5_Data2.累计热量小数, out => "RM5_累计热量")
   END_RUNG
   // the same network as SCL:
   "中间变量值".RM_TMP_REAL_1 := UDINT_TO_REAL("DB_MasterData".M1_Data2.累计热量整数);
   "RM1_累计热量" := "中间变量值".RM_TMP_REAL_1 + "DB_MasterData".M1_Data2.累计热量小数;
   "中间变量值".RM_TMP_REAL_2 := UDINT_TO_REAL("DB_MasterData".M2_Data2.累计热量整数);
   "RM2_累计热量" := "中间变量值".RM_TMP_REAL_2 + "DB_MasterData".M2_Data2.累计热量小数;
   "中间变量值".RM_TMP_REAL_3 := UDINT_TO_REAL("DB_MasterData".M3_Data2.累计热量整数);
   "RM3_累计热量" := "中间变量值".RM_TMP_REAL_3 + "DB_MasterData".M3_Data2.累计热量小数;
   "中间变量值".RM_TMP_REAL_4 := UDINT_TO_REAL("DB_MasterData".M4_Data2.累计热量整数);
   "RM4_累计热量" := "中间变量值".RM_TMP_REAL_4 + "DB_MasterData".M4_Data2.累计热量小数;
   "中间变量值".RM_TMP_REAL_5 := UDINT_TO_REAL("DB_MasterData".M5_Data2.累计热量整数);
   "RM5_累计热量" := "中间变量值".RM_TMP_REAL_5 + "DB_MasterData".M5_Data2.累计热量小数;
END_REGION

REGION Network 4: 入口温度
   // 入口温度
